(* CODESYS project TcDynCollections.library
   Company: FisoThemes
   DefaultNamespace: TcDynCollections
   Version: 1.0.5.27
   DocFormat: reStructuredText
   Placeholder: TwinCat Dynamic Collections
   Author: Goodwill Mzumala
   Description: A library for handling collections of data dynamically in TwinCAT.
   Title: TwinCat Dynamic Collections

Project tree, tasks and I/O mapping:
  libraries: Tc2_Standard, * (Beckhoff Automation GmbH); Tc2_System, * (Beckhoff Automation GmbH); Tc2_Utilities, 3.3.38.0 (Beckhoff Automation GmbH); Tc3_Module, * (Beckhoff Automation GmbH)
  DUTs/
    Aliases/
      data type T_AVL_Map_Node
      data type T_AVL_Node
      data type T_BST_Traversal
      data type T_Capacity
      data type T_Comparison
      data type T_Error
      data type T_Generic
      data type T_Hashmap_Bucket_Node
      data type T_Hashset_Bucket_Node
      data type T_List_Node
      data type T_Map_Entry
      data type T_Position
      data type T_Type
    Enums/
      data type E_BINARY_SEARCH_TREE_TRAVERSAL
      data type E_COMPARISON
      data type E_ERROR_CODE
    Structs/
      data type ST_AVL_MAP_NODE
      data type ST_AVL_NODE
      data type ST_ERROR
      data type ST_HASHMAP_BUCKET_NODE
      data type ST_HASHSET_BUCKET_NODE
      data type ST_LIST_NODE
      data type ST_MAP_ENTRY
      data type ST_ORDERED_HASHMAP_BUCKET_NODE
      data type ST_ORDERED_HASHSET_BUCKET_NODE
  GVLs/
    global variables GVL_Constants
    global variables GVL_Errors
  ITFs/
    Collections/
      Immutable/
        interface I_Immutable_Array: _Begin, _End, Contains, Get, Get_As_String, Get_Type_At, Search
        interface I_Immutable_Collection
        interface I_Immutable_List: _Begin, _End, Contains, Get, Get_As_String, Get_Type_At, Search
        interface I_Immutable_Map: Contains, Get, Get_As_String, Get_Keys, Get_Values
        interface I_Immutable_Set: Contains, Get_Values
      interface I_Array: _Begin, _End, Contains, Get, Get_As_String, Get_Generic, Get_Type_At, Reverse, Search, Set, Set_Generic, Swap
      interface I_Array_List: _Capacity
      interface I_Collection: _Count, _Empty, _Error_Status
      interface I_Deque: _Values, Back, Clear, Dequeue_At_Back, Dequeue_At_Front, Enqueue_At_Back, Enqueue_At_Front, Enqueue_Generic, Front, Reverse
      interface I_Hash_Map: _Bucket_Count, Resize
      interface I_Hash_Set: _Bucket_Count, Resize
      interface I_List: _Begin, _End, Append, Clear, Contains, Get, Get_As_String, Get_Generic, Get_Type_At, Insert, Insert_Generic, Prepend, Remove, Remove_At, Remove_Last, Resize, Reverse, Search, Set, Set_Generic, Swap
      interface I_Map: Clear, Contains, Get, Get_As_String, Get_Generic, Get_Keys, Get_Values, Insert, Insert_Generic, Remove, Remove_Generic, Update, Update_Generic, Upsert
      interface I_Queue: _Values, Clear, Dequeue, Enqueue, Enqueue_At_Front, Enqueue_Generic, Get, Get_Generic, Reverse
      interface I_Set: Clear, Contains, Get_Values, Insert, Insert_Generic, Remove, Remove_Generic
      interface I_Stack: _Values, Clear, Get, Get_Generic, Pop, Push, Push_Generic, Reverse
      interface I_Tree_Map: _Traversal
      interface I_Tree_Set: _Traversal
    Enumerators/
      interface I_Enumerable: Get_Enumerator
      interface I_Enumerator: Current, Current_As_String, Dispose, Next, Reset
    Iterable/
      interface I_Iterable: _Begin, _End
    Misc/
      interface I_Copyable: Copy_To
  POUs/
    Examples/
    Function Blocks/
      Collections/
        Immutable/
          function block FB_Immutable_Array [ST]: _Begin, _Count, _Empty, _End, _Error_Status, Contains, Get, Get_As_String, Get_Type_At, Search
          function block FB_Immutable_List [ST]: _Begin, _Count, _Empty, _End, _Error_Status, Contains, Get, Get_As_String, Get_Type_At, Search
          function block FB_Immutable_Map [ST]: _Count, _Empty, _Error_Status, Contains, Get, Get_As_String, Get_Keys, Get_Values
          function block FB_Immutable_Set [ST]: _Count, _Empty, _Error_Status, Contains, Get_Values
        function block FB_Array [ST]: _Begin, _End, Contains, FB_exit, FB_init, Get, Get_As_String, Get_Generic, Get_Type_At, Reverse, Search, Set, Set_Generic, Swap
        function block FB_Array_List [ST]: _Begin, _Capacity, _End, Append, Clear, Contains, FB_exit, FB_init, Get, Get_As_String, Get_Generic, Get_Type_At, Insert, Insert_Generic, Prepend, Remove, Remove_At, Remove_Last, Resize, Reverse, Search, Set, Set_Generic, Swap
        function block FB_Collection [ST]: Clear_Error, Decrement_Count, Increment_Count, _Count, _Empty, _Error_Status
        function block FB_Deque [ST]: _Count, _Empty, _Error_Status, _Values, Back, Clear, Dequeue_At_Back, Dequeue_At_Front, Enqueue_At_Back, Enqueue_At_Front, Enqueue_Generic, Front, Reverse
        function block FB_Hash_Map [ST]: Create_Buckets, Create_Node, Delete_Node, Hash, _Bucket_Count, Clear, Contains, FB_exit, FB_init, Get, Get_As_String, Get_Generic, Get_Keys, Get_Values, Insert, Insert_Generic, Remove, Remove_Generic, Resize, Update, Update_Generic, Upsert
        function block FB_Hash_Set [ST]: Create_Buckets, Create_Node, Delete_Node, Hash, _Bucket_Count, Clear, Contains, FB_exit, FB_init, Get_Values, Insert, Insert_Generic, Remove, Remove_Generic, Resize
        function block FB_List [ST]: Closest_Node_Iterator, Iterate, _Begin, _End, Append, Clear, Contains, FB_exit, Get, Get_As_String, Get_Generic, Get_Type_At, Insert, Insert_Generic, Prepend, Remove, Remove_At, Remove_Last, Resize, Reverse, Search, Set, Set_Generic, Swap
        function block FB_Queue [ST]: _Count, _Empty, _Error_Status, _Values, Clear, Dequeue, Enqueue, Enqueue_At_Front, Enqueue_Generic, Get, Get_Generic, Reverse
        function block FB_Stack [ST]: _Count, _Empty, _Error_Status, _Values, Clear, Get, Get_Generic, Pop, Push, Push_Generic, Reverse
        function block FB_Tree_Map [ST]: Balance, Clear_Node, Create_Node, Delete_Node, Find_Minimum_Node, Get_Balance, Get_Height, Move_Node, Remove_Node, Rotate_Left, Rotate_Right, Search_Node, Update_Height, _Traversal, Clear, Contains, FB_exit, Get, Get_As_String, Get_Generic, Get_Keys, Get_Values, Insert, Insert_Generic, Remove, Remove_Generic, Update, Update_Generic, Upsert
        function block FB_Tree_Multiset [ST]: Insert_Generic
        function block FB_Tree_Set [ST]: Balance, Clear_Node, Create_Node, Delete_Node, Find_Minimum_Node, Get_Balance, Get_Height, Move_Node, Remove_Node, Rotate_Left, Rotate_Right, Search_Node, Update_Height, _Traversal, Clear, Contains, FB_exit, Get_Values, Insert, Insert_Generic, Remove, Remove_Generic
      Enumerators/
        function block FB_Enumerator [ST]: Current, Current_As_String, Dispose, FB_exit, FB_init, Next, Reset
      Misc/
        function block FB_Free [ST]: FB_exit, FB_init
      Specialised/
      Wrappers/
    Functions/
      function F_Any_To_Generic [ST]
      function F_Clone_Generic [ST]
      function F_Compare_Any [ST]
      function F_Compare_Generics [ST]
      function F_Copy_Generic_Value [ST]
      function F_Delete_Generic [ST]
      function F_Error [ST]
      function F_Generic_To_DT [ST]
      function F_Generic_To_LREAL [ST]
      function F_Generic_To_LTIME [ST]
      function F_Generic_To_String [ST]
      function F_Is_Date_Generic [ST]
      function F_Is_Numeric_Generic [ST]
      function F_Is_Time_Generic [ST]
      function F_Malloc_Generic [ST]
      function F_Matching_Generics [ST]
      function F_Murmur_Scramble [ST]
      function F_Murmur3_Hash [ST]
      function F_String_Convertable_Generic [ST]
      function F_String_To_Any [ST]
      function F_Swap_Generics [ST]
    program MAIN [ST]
  Project Information/
    function F_GetCompany [ST]
    function F_GetTitle [ST]
    function F_GetVersion [ST]
  UML/
    Collections Interfaces
  Version/
    global variables Global_Version
  VISUs/
*)

// DUTs/Aliases/T_AVL_Map_Node
TYPE T_AVL_Map_Node : ST_AVL_MAP_NODE; END_TYPE

// DUTs/Aliases/T_AVL_Node
TYPE T_AVL_Node : ST_AVL_NODE; END_TYPE

// DUTs/Aliases/T_BST_Traversal
TYPE T_BST_Traversal : E_BINARY_SEARCH_TREE_TRAVERSAL; END_TYPE

// DUTs/Aliases/T_Capacity
TYPE T_Capacity : DINT(GVL_Constants.MIN_CAPACITY..GVL_Constants.MAX_CAPACITY); END_TYPE

// DUTs/Aliases/T_Comparison
TYPE T_Comparison : E_COMPARISON; END_TYPE

// DUTs/Aliases/T_Error
TYPE T_Error : ST_ERROR; END_TYPE

// DUTs/Aliases/T_Generic
TYPE T_Generic : __SYSTEM.AnyType; END_TYPE

// DUTs/Aliases/T_Hashmap_Bucket_Node
TYPE T_Hashmap_Bucket_Node : ST_HASHMAP_BUCKET_NODE; END_TYPE

// DUTs/Aliases/T_Hashset_Bucket_Node
TYPE T_Hashset_Bucket_Node : ST_HASHSET_BUCKET_NODE; END_TYPE

// DUTs/Aliases/T_List_Node
TYPE T_List_Node : ST_LIST_NODE; END_TYPE

// DUTs/Aliases/T_Map_Entry
TYPE T_Map_Entry : ST_MAP_ENTRY; END_TYPE

// DUTs/Aliases/T_Position
TYPE T_Position : DINT; END_TYPE

// DUTs/Aliases/T_Type
TYPE T_Type : __SYSTEM.TYPE_CLASS; END_TYPE

// DUTs/Enums/E_BINARY_SEARCH_TREE_TRAVERSAL
// Methods for traversing a binary search tree.
{attribute 'qualified_only'}
{attribute 'to_string'}
TYPE E_BINARY_SEARCH_TREE_TRAVERSAL :
(
	In_Order := 0,
	Pre_Order,
	Post_Order, 
	Level_Order
)BYTE;
END_TYPE

// DUTs/Enums/E_COMPARISON
// Comparison enum.
{attribute 'qualified_only'}
{attribute 'strict'}
{attribute 'to_string'}
TYPE E_COMPARISON :
(
	Invalid := 0,
	Less,
	Equal,
	Greater
)BYTE;
END_TYPE

// DUTs/Enums/E_ERROR_CODE
 // Error code are @ CmpErrors.Errors.<variable> from the CmpErrors2 Interfaces library.
 // https://help.codesys.com/webapp/Errors;product=CmpErrors2_Itfs;version=3.5.15.0
{attribute 'qualified_only'}
{attribute 'to_string'}
TYPE E_ERROR_CODE :
(
	ERR_OK 						 := 16#0,	//	Ok
	ERR_FAILED 					 := 16#1, 	//	General error - To be used only for internal errors
	ERR_PARAMETER 				 := 16#2, 	//	Invalid parameter for this operation
	ERR_NOT_INITIALIZED 		 := 16#3, 	//	Function cannot be executed, since component has not been initialized yet. It may work later, though
	ERR_VERSION 				 := 16#4, 	//	Version conflict
	ERR_TIMEOUT 				 := 16#5, 	//	Operation timed out
	ERR_NO_BUFFER 				 := 16#6, 	//	Insufficient memory to carry out the request
	ERR_PENDING 				 := 16#A, 	//	For async-calls: call not complete, yet
	ERR_NUM_PENDING 			 := 16#B, 	//  Too many pending calls. Try later
	ERR_NOT_IMPLEMENTED 		 := 16#C, 	//  The function is not implemented
	ERR_INVALID_ID 				 := 16#D, 	//  No object with the provided id found
	ERR_OVERFLOW 				 := 16#E, 	//	Integer overflow
	ERR_BUFFER_SIZE 			 := 16#F, 	//	The size of a buffer is too small OR invalid
	ERR_NO_OBJECT 				 := 16#10,	//	No object with this specified name available
	ERR_NO_MEMORY 				 := 16#11,	//  No heap memory available
	ERR_DUPLICATE 				 := 16#12A, //  An object with the same name is still available
	ERR_MEMORY_OVERWRITE 		 := 16#13,  //  Heap memory was written out of bounds! Memory overwrite error
	ERR_INVALID_HANDLE 			 := 16#14,  //  Invalid handle to an object
	ERR_END_OF_0BJECT 			 := 16#15,  //  End OF object reached
	ERR_NO_CHANGE 				 := 16#16,  //  No changes done
	ERR_INVALID_INTERFACE 		 := 16#17,  //  Invalid or unknown interface
	ERR_NOT_SUPPORTED 			 := 16#18,  //  Functionality not supported
	ERR_NO_ACCESS_RIGHTS 		 := 16#19,  //  No access rights for this operation
	ERR_OUT_OF_LIMITS 			 := 16#1A,  //  Specified limits of a resource exceeded
	ERR_ENTRIES_REMAINING 		 := 16#1B,  //  Remaining entries that could not be transmitted because of buffer limitation
	ERR_INVALID_SESSION_ID 		 := 16#1C,  //  Invalid online sessionid
	ERR_EXCEPTION 				 := 16#1D,  //  Exception occurred
	ERR_SIGNATURE_MISMATCH 		 := 16#1E,	//	Signature mismatch of an api function
	ERR_VERSION_MISMATCH 		 := 16#1F,	//	Version mismatch
	ERR_TYPE_MISMATCH 			 := 16#20,	//	Type mismatch
	ERR_ID_MISMATCH 			 := 16#21,	//	ID mismatch
	ERR_NO_CONSISTENCY 			 := 16#22,	//	Consistency error
	ERR_NO_COMM_CYCLE 			 := 16#23,	//	No COMM_CYCLE needed
	ERR_DONT_SUSPEND_TASK 		 := 16#24,	//	Do not suspend task after an exception
	ERR_MEMORY_LOCK_FAILED 		 := 16#25,	//	Memory cannot be locked in this operation
	ERR_LICENSE_MISSING 		 := 16#26,	//	License missing for the runtime
	ERR_OPERATION_DENIED 		 := 16#27,	//	Operation denied 
	ERR_DEVICE 					 := 16#28,	//	Device error
	ERR_DISK_FULL 				 := 16#29,	//	Disk full
	ERR_CRC_FAILED 				 := 16#30,	//	Internal use in runtime
	ERR_MEDIA_ERASE 			 := 16#31,	//	Internal use in runtime
	ERR_FILE_ERROR 				 := 16#32,	//	File error. e.g. cannot open a file for writing because it could be write protected
	ERR_NO_RETAIN_MEMORY 		 := 16#33,	//	No retain memory available
	ERR_OUT_OF_LIMITS_MIN 		 := 16#34,	//	Specified minimum-limit of a resource exceeded
	ERR_OUT_OF_LIMITS_MAX 		 := 16#35,	//	Specified maximum-limit of a resource exceeded
	ERR_SIZE_MISMATCH 			 := 16#36,	//	Size mismatch
	ERR_CALL_AGAIN 				 := 16#37,	//	Operation is not yet finished, call function again to proceed
	ERR_NOTHING_TO_DO 			 := 16#38,	//	Operation has nothing to do. No execution.
	ERR_SECURITY_CHECKS_FAILED 	 := 16#39,	//	Some security checks have failed. /* This is a generic error code to report this error over public channels. In this case the error code doesn’t provide a detailed cause for the error. */
	ERR_INVALID_SEQUENCE 		 := 16#3A,	//	 
	ERR_INVALID_REFERENCE 		 := 16#3B,	//	Dereferencing an IEC reference in IecVarAccess failed due to invalid destination address, e. G. NULL.
	ERR_CONVERSION_INCOMPLETE 	 := 16#3C,	//	Conversion of string encodings was not lossless.
	ERR_SOCK_NOT_INITIALIZED 	 := 16#201, //  Socket errors (range: 0x0200 - 0X02FF)
	ERR_SOCK_NOT_SOCKET 		 := 16#202, //  The provided socket handle is invalid
	ERR_SOCK_AF_UNSUPPORTED 	 := 16#203, //  The address family is not supported
	ERR_SOCK_PROTO_UNSUPPORTED   := 16#204, //  Protocol is not supported */
	ERR_SOCK_NO_BUFFER 			 := 16#205, //  Not enough buffer to handle the request */
	ERR_SOCK_WOULD_BLOCK 		 := 167206, //  Socket is in nonblocking mode but this call would block =/
	ERR_SOCK_ADDR_INUSE 		 := 16#207, //  The provided address is already in use */
	ERR_SOCK_ADDR_NOT_AVAILABLE  := 16#208, //  The provided address is not available on THIS computer */
	ERR_SOCK_CONN_REFUSED 		 := 16#209, //  Connection has been refused by the remote host */
	ERR_SOCK_TIMEDOUT 			 := 16#20A, //  Operation timed out */
	ERR_SOCK_HOST_NOT_FOUND 	 := 16#20B, //  The host has NOT been found */
	ERR_SOCK_HOST_UNREACHABLE  	 := 16#20C, //  Host is unreachable */
	ERR_SOCK_1S_CONNECTED 		 := 16#20D, //  Socket is already connected =/
	ERR_SOCK_NOT_CONNECTED 		 := 16#20E, //  The socket is not connected */
	ERR_SOCK_SHUTDOWN 			 := 16#20F, //  Shutdown has been called on the socket =/
	ERR_SOCK_MSGSIZE 			 := 16#210, //  For sockets of type DGRAM. The package to send exceeds the maximum package size =/
	ERR_SOCK_CLOSED 			 := 16#211, //  Socket has been gracefully closed. No more send/receives allowed =/
	ERR_L7_TAG_MISSING 			 := 16#300,	//  Tag missing in online communication buffer
	ERR_L7_UNKNOWN_CMD_GROUP 	 := 16#301,	//  Unknown command group
	ERR_L7_UNKNOWN_CMD 			 := 16#302,	//  Unknown command (within a valid command group)
	ERR_L7_INCOMPLETE 			 := 16#303	//  Level 7 service incomplete
)DINT;
END_TYPE

// DUTs/Structs/ST_AVL_MAP_NODE
// Node for an AVL Tree Map.
{attribute 'enable_dynamic_creation'}
TYPE ST_AVL_MAP_NODE EXTENDS ST_MAP_ENTRY :
STRUCT
	Height 		: T_Position; // Height of the node.
	pParent 	: POINTER TO ST_AVL_MAP_NODE; 	// Pointer to parent node.
	pLeft 		: POINTER TO ST_AVL_MAP_NODE; 	// Pointer to left node.
	pRight 		: POINTER TO ST_AVL_MAP_NODE; 	// Pointer to right node.
END_STRUCT
END_TYPE

// DUTs/Structs/ST_AVL_NODE
// Node for AVL Tree.
{attribute 'enable_dynamic_creation'}
TYPE ST_AVL_NODE:
STRUCT
	Data 		: T_Generic; // Stored data.
	Height 		: T_Position; // Height of the node.
	pParent 	: POINTER TO ST_AVL_NODE; 	// Pointer to parent node.
	pLeft 		: POINTER TO ST_AVL_NODE; 	// Pointer to left node.
	pRight 		: POINTER TO ST_AVL_NODE; 	// Pointer to right node.
END_STRUCT
END_TYPE

// DUTs/Structs/ST_ERROR
// STRUCT used to contain error status information.
{attribute 'enable_dynamic_creation'}
TYPE ST_ERROR :
STRUCT
	nCODE 	: DINT; // Error code specific to the particular error.
	bSTATUS : BOOL; // Indicates if an error has occurred | TRUE = error, FALSE = no error
	sSOURCE : STRING; // Textual information describing the error.
END_STRUCT
END_TYPE

// DUTs/Structs/ST_HASHMAP_BUCKET_NODE
{attribute 'enable_dynamic_creation'}
TYPE ST_HASHMAP_BUCKET_NODE EXTENDS ST_MAP_ENTRY :
STRUCT
	pNext : POINTER TO ST_HASHMAP_BUCKET_NODE;
END_STRUCT
END_TYPE

// DUTs/Structs/ST_HASHSET_BUCKET_NODE
{attribute 'enable_dynamic_creation'}
TYPE ST_HASHSET_BUCKET_NODE :
STRUCT
	Data : T_Generic;
	pNext : POINTER TO ST_HASHSET_BUCKET_NODE;
END_STRUCT
END_TYPE

// DUTs/Structs/ST_LIST_NODE
// Node for linked list.
{attribute 'enable_dynamic_creation'}
TYPE ST_LIST_NODE:
STRUCT
	Data 		: T_Generic; // Stored data.
	pPrevious 	: POINTER TO ST_LIST_NODE; 	// Pointer to previous node.
	pNext 		: POINTER TO ST_LIST_NODE; 	// Pointer to next node.
END_STRUCT
END_TYPE

// DUTs/Structs/ST_MAP_ENTRY
// Entry for a key value pair.
{attribute 'enable_dynamic_creation'}
TYPE ST_MAP_ENTRY :
STRUCT
	Key : T_Generic; // Key used to identify stored value    
	Value : T_Generic; // Value to store in dictionary with key
END_STRUCT
END_TYPE

// DUTs/Structs/ST_ORDERED_HASHMAP_BUCKET_NODE
{attribute 'enable_dynamic_creation'}
TYPE ST_ORDERED_HASHMAP_BUCKET_NODE EXTENDS ST_MAP_ENTRY:
STRUCT
	pNext,
	pBefore,
	pAfter 	: POINTER TO ST_ORDERED_HASHSET_BUCKET_NODE;
END_STRUCT
END_TYPE

// DUTs/Structs/ST_ORDERED_HASHSET_BUCKET_NODE
{attribute 'enable_dynamic_creation'}
TYPE ST_ORDERED_HASHSET_BUCKET_NODE :
STRUCT
	Data 	: T_Generic;
	pNext,
	pBefore,
	pAfter 	: POINTER TO ST_ORDERED_HASHSET_BUCKET_NODE;
END_STRUCT
END_TYPE

// GVLs/GVL_Constants
{attribute 'qualified_only'}
VAR_GLOBAL CONSTANT
	MIN_CAPACITY : DINT := 0;
	MAX_CAPACITY : DINT := 2147483647;
END_VAR

// GVLs/GVL_Errors
// Library errors
{attribute 'qualified_only'}
VAR_GLOBAL CONSTANT
	ERR_NO_ERROR 			: T_Error := (bStatus := FALSE,	nCode := E_ERROR_CODE.ERR_OK, 				sSource := 'No Error.'); // No Error.
	ERR_TYPE_MISMATCH 		: T_Error := (bStatus := TRUE,	nCode := E_ERROR_CODE.ERR_TYPE_MISMATCH, 	sSource := 'Type mismatch.'); // Type mismatch.
	ERR_SIZE_MISMATCH 		: T_Error := (bStatus := TRUE,	nCode := E_ERROR_CODE.ERR_SIZE_MISMATCH, 	sSource := 'Size mismatch.'); // Size mismatch.
	ERR_INVALID_REFERENCE 	: T_Error := (bStatus := TRUE,	nCode := E_ERROR_CODE.ERR_INVALID_REFERENCE,sSource := 'Invalid reference.'); // Invalid reference.
	ERR_INVALID_INTERFACE 	: T_Error := (bStatus := TRUE,	nCode := E_ERROR_CODE.ERR_INVALID_INTERFACE,sSource := 'Invalid interface.'); // Invalid interface.
	ERR_INVALID_CONVERSION	: T_Error := (bStatus := TRUE,	nCode := E_ERROR_CODE.ERR_NOT_SUPPORTED, 	sSource := 'Conversion not supported.'); // Conversion not supported.
	ERR_INVALID_COMPARISON	: T_Error := (bStatus := TRUE,	nCode := E_ERROR_CODE.ERR_NOT_SUPPORTED, 	sSource := 'Invalid comparison.'); // Invalid comparison.
	ERR_NO_KEY 				: T_Error := (bStatus := TRUE,	nCode := E_ERROR_CODE.ERR_NO_OBJECT,		sSource := 'Key not found.'); // Key not found.'
	ERR_NO_ITEM 			: T_Error := (bStatus := TRUE,	nCode := E_ERROR_CODE.ERR_NO_OBJECT, 		sSource := 'Item not found.'); // Item not found.
	ERR_INDEX_OUT_OF_BOUNDS : T_Error := (bStatus := TRUE,	nCode := E_ERROR_CODE.ERR_OUT_OF_LIMITS, 	sSource := 'Index out of bounds.'); // Index out of bounds.
	ERR_DUPLICATE_KEY 		: T_Error := (bStatus := TRUE,	nCode := E_ERROR_CODE.ERR_DUPLICATE, 		sSource := 'Duplicate key.'); // Duplicate key.
	ERR_DUPLICATE_ITEM 		: T_Error := (bStatus := TRUE,	nCode := E_ERROR_CODE.ERR_DUPLICATE, 		sSource := 'Duplicate item.'); // Duplicate item.
	ERR_MALLOC_FAILED 		: T_Error := (bStatus := TRUE,	nCode := E_ERROR_CODE.ERR_NO_MEMORY, 		sSource := 'Memory allocation failed.'); // Memory allocation failed.
END_VAR

// Version/Global_Version
{attribute 'TcGenerated'}
{attribute 'no-analysis'}
{attribute 'linkalways'}
// This function has been automatically generated from the project information.
VAR_GLOBAL CONSTANT
	{attribute 'const_non_replaced'}
	stLibVersion_TwinCat_Dynamic_Collections : ST_LibVersion := (iMajor := 1, iMinor := 0, iBuild := 5, iRevision := 27, nFlags := 0, sVersion := '1.0.5.27');
END_VAR

// ITFs/Collections/Immutable/I_Immutable_Array
// Interface for an immutable array.
INTERFACE I_Immutable_Array EXTENDS I_Immutable_Collection

// Index of the first element.
PROPERTY _Begin : T_Position
GET
END_GET
END_PROPERTY

// Index of the last element.
PROPERTY _End : T_Position
GET
END_GET
END_PROPERTY

// Checks if item is contained in array.
METHOD Contains : BOOL
VAR_INPUT
	Item : ANY; // Item to find.
END_VAR
END_METHOD

// Gets item from array at specified location.
METHOD Get : I_Immutable_Array
VAR_INPUT
	Index : T_Position; // Location of item.
	Item : ANY;  // Variable to store returned item.
END_VAR
VAR_OUTPUT
	bSuccess : BOOL;
END_VAR
END_METHOD

// Returns item as a string, if type to string conversion is supported.
METHOD Get_As_String : I_Immutable_Array
VAR_INPUT
	Index : T_Position; // Location of item.
	sItem : REFERENCE TO STRING; // Variable to store returned item.
END_VAR
VAR_OUTPUT
	bSuccess : BOOL;
END_VAR
END_METHOD

// Gets the type of the item at specified location.
METHOD Get_Type_At : I_Immutable_Array
VAR_INPUT
	Index : T_Position;
END_VAR
VAR_OUTPUT
	Item_Type : T_Type;
	bSuccess : BOOL;
END_VAR
END_METHOD

// Find the location of an item in the array.
METHOD Search : I_Immutable_Array
VAR_INPUT
	Item : ANY; // Item to find.
END_VAR
VAR_OUTPUT
	Index : T_Position; //Location of item.
	bSuccess : BOOL;
END_VAR
END_METHOD

END_INTERFACE

// ITFs/Collections/Immutable/I_Immutable_Collection
// Base interface for immutable collections
INTERFACE I_Immutable_Collection EXTENDS I_Collection

END_INTERFACE

// ITFs/Collections/I_Collection
// Base interface for collections.
INTERFACE I_Collection EXTENDS __SYSTEM.IQueryInterface

// Number of items in the collection.
PROPERTY _Count : T_Capacity
GET
END_GET
END_PROPERTY

// Checks if collection is empty.
PROPERTY _Empty : BOOL
GET
END_GET
END_PROPERTY

// Error status of the collection.
PROPERTY _Error_Status : T_Error
GET
END_GET
END_PROPERTY

END_INTERFACE

// ITFs/Collections/Immutable/I_Immutable_List
// Interface for an immutable list.
INTERFACE I_Immutable_List EXTENDS I_Immutable_Collection

// Index of the first element.
PROPERTY _Begin : T_Position
GET
END_GET
END_PROPERTY

// Index of the last element.
PROPERTY _End : T_Position
GET
END_GET
END_PROPERTY

(* Checks if item is contained in list *)
METHOD Contains : BOOL
VAR_INPUT
	Item : ANY; // Item to find in list
END_VAR
END_METHOD

// Gets item from list at specified location without removing it.
METHOD Get : I_Immutable_List
VAR_INPUT
	Index : T_Position; // Location of item
	Item : ANY;  // Variable to store returned item
END_VAR
VAR_OUTPUT
	bSuccess : BOOL;
END_VAR
END_METHOD

// Returns item as a string, if type to string conversion is supported.
METHOD Get_As_String : I_Immutable_List
VAR_INPUT
	Index : T_Position; // Location of item
	sItem : REFERENCE TO STRING; // Variable to store returned item.
END_VAR
VAR_OUTPUT
	bSuccess : BOOL;
END_VAR
END_METHOD

// Gets the type of the item at specified location.
METHOD Get_Type_At : I_Immutable_List
VAR_INPUT
	Index : T_Position;
END_VAR
VAR_OUTPUT
	Item_Type : T_Type;
	bSuccess : BOOL;
END_VAR
END_METHOD

// Find the location of an item in list.
METHOD Search : I_Immutable_List
VAR_INPUT
	Item : ANY; // Item to find in list
END_VAR
VAR_OUTPUT
	Index : T_Position; //Location of item in list 
	bSuccess : BOOL;
END_VAR
END_METHOD

END_INTERFACE

// ITFs/Collections/Immutable/I_Immutable_Map
INTERFACE I_Immutable_Map EXTENDS I_Immutable_Collection

// Checks if key is contained in the map.
METHOD Contains : BOOL
VAR_INPUT
	Key : ANY; // Key to find.
END_VAR
END_METHOD

// Gets the value associated with the specified key without removing it from the map.
METHOD Get : I_Immutable_Map
VAR_INPUT
	Key : ANY; // Key used to identify stored value
	Value : ANY; // Variable to store requested data 
END_VAR
VAR_OUTPUT
	bSuccess : BOOL;
END_VAR
END_METHOD

// Returns value as a string, if type to string conversion is supported.
METHOD Get_As_String : I_Immutable_Map
VAR_INPUT
	Key : ANY; // Key used to identify stored value
	sValue : REFERENCE TO STRING; // Variable to store returned item.
END_VAR
VAR_OUTPUT
	bSuccess : BOOL;
END_VAR
END_METHOD

// Gets an immutable list of the keys.
METHOD Get_Keys : I_Immutable_List
VAR_INPUT
END_VAR
END_METHOD

// Gets an immutable list of the values.
METHOD Get_Values : I_Immutable_List
VAR_INPUT
END_VAR
END_METHOD

END_INTERFACE

// ITFs/Collections/Immutable/I_Immutable_Set
// Interface for immutable set.
INTERFACE I_Immutable_Set EXTENDS I_Immutable_Collection

// Checks if item is contained in set.
METHOD Contains : BOOL
VAR_INPUT
	Item : ANY; // Item to find.
END_VAR
END_METHOD

// Gets an immutable list of the values in the set.
METHOD Get_Values : I_Immutable_List
END_METHOD

END_INTERFACE

// ITFs/Collections/I_Array
// Interface for a static array.
INTERFACE I_Array EXTENDS I_Collection

// Index of the first element.
PROPERTY _Begin : T_Position
GET
END_GET
END_PROPERTY

// Index of the last element.
PROPERTY _End : T_Position
GET
END_GET
END_PROPERTY

// Checks if item is contained in array.
METHOD Contains : BOOL
VAR_INPUT
	Item : ANY; // Item to find.
END_VAR
END_METHOD

// Gets item from array at specified location.
METHOD Get : I_Array
VAR_INPUT
	Index : T_Position; // Location of item.
	Item : ANY;  // Variable to store returned item.
END_VAR
VAR_OUTPUT
	bSuccess : BOOL;
END_VAR
END_METHOD

// Returns item as a string, if type to string conversion is supported.
METHOD Get_As_String : I_Array
VAR_INPUT
	Index : T_Position; // Location of item.
	sItem : REFERENCE TO STRING; // Variable to store returned item.
END_VAR
VAR_OUTPUT
	bSuccess : BOOL;
END_VAR
END_METHOD

// Gets an item from the array in it's generic form.
// (** Use carefully as this contains the pointer of the actual value in the collection. **)
// If you wish to use this it is recommeded you create a copy of the returned value using MEMMOVE or MEMCPY
METHOD Get_Generic : I_Array
VAR_INPUT
	Index : T_Position; // Location of item.
END_VAR
VAR_OUTPUT
	Item : T_Generic;
	bSuccess : BOOL;
END_VAR
END_METHOD

// Gets the type of the item at specified location.
METHOD Get_Type_At : I_Array
VAR_INPUT
	Index : T_Position;
END_VAR
VAR_OUTPUT
	Item_Type : T_Type;
	bSuccess : BOOL;
END_VAR
END_METHOD

// Reverses the order of items in the array.
METHOD Reverse : I_Array
VAR_OUTPUT
	bSuccess : BOOL;
END_VAR
END_METHOD

// Find the location of an item in the array.
METHOD Search : I_Array
VAR_INPUT
	Item : ANY; // Item to find.
END_VAR
VAR_OUTPUT
	Index : T_Position; //Location of item.
	bSuccess : BOOL;
END_VAR
END_METHOD

// Changes the item at the specified location in the array.
METHOD Set : I_Array
VAR_INPUT
	Index 	: T_Position; // Location of item.
	Item 	: ANY; 	// Item to store.
END_VAR
VAR_OUTPUT
	bSuccess : BOOL;
END_VAR
END_METHOD

// Changes the item at the specified location in the array in it's generic form.
METHOD Set_Generic : I_Array
VAR_INPUT
	Index : T_Position; // Location of item.
	Item : T_Generic; // Item to store.
END_VAR
VAR_OUTPUT
	bSuccess : BOOL;
END_VAR
END_METHOD

// Swaps item at index with item at index B.
METHOD Swap : I_Array
VAR_INPUT
	Index_A, Index_B : T_Position;
END_VAR
VAR_OUTPUT
	bSuccess : BOOL;
END_VAR
END_METHOD

END_INTERFACE

// ITFs/Collections/I_Array_List
// Interface for the array list.
INTERFACE I_Array_List EXTENDS I_List

// Size of the storage space currently allocated for the array list.
PROPERTY _Capacity : T_Capacity
GET
END_GET
END_PROPERTY

END_INTERFACE

// ITFs/Collections/I_List
// Interface for a list.
INTERFACE I_List EXTENDS I_Collection

// Index of the first element.
PROPERTY _Begin : T_Position
GET
END_GET
END_PROPERTY

// Index of the last element.
PROPERTY _End : T_Position
GET
END_GET
END_PROPERTY

// Adds an item to the end of the list.
METHOD Append : I_List
VAR_INPUT
	Item : ANY; // Value to store in list
END_VAR
VAR_OUTPUT
	bSuccess : BOOL;
END_VAR
END_METHOD

// Empties/Clears/Deletes every item in the list.
METHOD Clear : I_List
END_METHOD

// Checks if item is contained in list.
METHOD Contains : BOOL
VAR_INPUT
	Item : ANY; // Item to find in list
END_VAR
END_METHOD

// Gets item from list at specified location without removing it
METHOD Get : I_List
VAR_INPUT
	Index : T_Position; // Location of item
	Item : ANY;  // Variable to store returned item
END_VAR
VAR_OUTPUT
	bSuccess : BOOL;
END_VAR
END_METHOD

// Returns item as a string, if type to string conversion is supported
METHOD Get_As_String : I_List
VAR_INPUT
	Index : T_Position; // Location of item
	sItem : REFERENCE TO STRING; // Variable to store returned item.
END_VAR
VAR_OUTPUT
	bSuccess : BOOL;
END_VAR
END_METHOD

// Gets a value from a list in it's generic form.
// (** Use carefully as this contains the pointer of the actual value in the collection. **)
// If you wish to use this it is recommeded you create a copy of the returned value using MEMMOVE or MEMCPY
METHOD Get_Generic : I_List
VAR_INPUT
	Index : T_Position; // Location of item
END_VAR
VAR_OUTPUT
	Item : T_Generic;
	bSuccess : BOOL;
END_VAR
END_METHOD

// Gets the type of the item at specified location.
METHOD Get_Type_At : I_List
VAR_INPUT
	Index : T_Position;
END_VAR
VAR_OUTPUT
	Item_Type : T_Type;
	bSuccess : BOOL;
END_VAR
END_METHOD

// Adds new item to list at specified location, if index = 0, item will be added at the front, if index = count, item will be added at the back
METHOD Insert : I_List
VAR_INPUT
	Index : T_Position; // Location of item
	Item : ANY; // Item to store in list
END_VAR
VAR_OUTPUT
	bSuccess : BOOL;
END_VAR
END_METHOD

// Adds new item to list at specified location using the generic form. 
// If index = 0, item will be added at the front, if index = count, item will be added at the back
METHOD Insert_Generic : I_List
VAR_INPUT
	Index 	 : T_Position; 	// Location of item
	Item 	 : T_Generic;  	// Item to store in list
END_VAR
VAR_OUTPUT
	bSuccess : BOOL;
END_VAR
END_METHOD

// Adds an item at the front of the list.
METHOD Prepend : I_List
VAR_INPUT
	Item : ANY; // Value to store in list
END_VAR
VAR_OUTPUT
	bSuccess : BOOL;
END_VAR
END_METHOD

// Removes item from the list.
METHOD Remove : I_List
VAR_INPUT
	Item : ANY; // Item to remove from in list
END_VAR
VAR_OUTPUT
	bSuccess : BOOL;
END_VAR
END_METHOD

// Remove item at specified location 
METHOD Remove_At : I_List
VAR_INPUT
	Index : T_Position; // Location of item
END_VAR
VAR_OUTPUT
	bSuccess : BOOL;
END_VAR
END_METHOD

// Removes item at the back of the list.
METHOD Remove_Last : I_List
VAR_OUTPUT
	bSuccess : BOOL;
END_VAR
END_METHOD

// Manually resize list. If list becomes smaller, item on higher locations will be deleted.
METHOD Resize : I_List
VAR_INPUT
	Size : T_Capacity; // New size of list.
END_VAR
VAR_OUTPUT
	bSuccess : BOOL;
END_VAR
END_METHOD

// Reverses the order of items in the list
METHOD Reverse : I_List
VAR_OUTPUT
	bSuccess : BOOL;
END_VAR
END_METHOD

// Find the location of an item in list.
METHOD Search : I_List
VAR_INPUT
	Item : ANY; // Item to find in list
END_VAR
VAR_OUTPUT
	Index : T_Position; //Location of item in list 
	bSuccess : BOOL;
END_VAR
END_METHOD

// Changes the item at the specified location in the list.
METHOD Set : I_List
VAR_INPUT
	Index 	: T_Position; // Location of item
	Item 	: ANY; 	// Item to store in list
END_VAR
VAR_OUTPUT
	bSuccess : BOOL;
END_VAR
END_METHOD

// Changes the item at the specified location in the list in it's generic form.
METHOD Set_Generic : I_List
VAR_INPUT
	Index : T_Position; // Location of item
	Item : T_Generic; // Item to store in list
END_VAR
VAR_OUTPUT
	bSuccess : BOOL;
END_VAR
END_METHOD

// Swaps item at index A with item at index B.
METHOD Swap : I_List
VAR_INPUT
	Index_A, Index_B : T_Position;
END_VAR
VAR_OUTPUT
	bSuccess : BOOL;
END_VAR
END_METHOD

END_INTERFACE

// ITFs/Collections/I_Deque
// Interface for a double ended queue - Deque
INTERFACE I_Deque EXTENDS I_Collection

// Gets an immutable list of the items in Deque.
PROPERTY _Values : I_Immutable_List
GET
END_GET
END_PROPERTY

// Get item at the back of the deque without removing it.
METHOD Back : I_Deque
VAR_INPUT
	Item : ANY; // Variable to store returned item value
END_VAR
VAR_OUTPUT
	bSuccess : BOOL;
END_VAR
END_METHOD

// Empties/Clears/Deletes every item in the deque.
METHOD Clear : I_Deque
END_METHOD

// Removes item at the front of the deque.
METHOD Dequeue_At_Back : I_Deque
VAR_OUTPUT
	bSuccess : BOOL;
END_VAR
END_METHOD

// Removes item at the front of the deque.
METHOD Dequeue_At_Front : I_Deque
VAR_OUTPUT
	bSuccess : BOOL;
END_VAR
END_METHOD

// Adds item at the back of the deque.
METHOD Enqueue_At_Back : I_Deque
VAR_INPUT
	Item : ANY; // Item to store.
END_VAR
VAR_OUTPUT
	bSuccess : BOOL;
END_VAR
END_METHOD

// Add item to the front of the deque.
METHOD Enqueue_At_Front : I_Deque
VAR_INPUT
	Item : ANY; // Item to store.
END_VAR
VAR_OUTPUT
	bSuccess : BOOL;
END_VAR
END_METHOD

// Adds a generic item at the back of the deque.
METHOD Enqueue_Generic : I_Deque
VAR_INPUT
	Item : T_Generic; // Item to store.
	bAt_Front : BOOL; // Enqueues at front if set to TRUE.
END_VAR
VAR_OUTPUT
	bSuccess : BOOL;
END_VAR
END_METHOD

// Get item at the front of the deque without removing it.
METHOD Front : I_Deque
VAR_INPUT
	Item : ANY; // Variable to store returned item value
END_VAR
VAR_OUTPUT
	bSuccess : BOOL;
END_VAR
END_METHOD

// Reverses the order of items in the deque.
METHOD Reverse : I_Deque
VAR_OUTPUT
	bSuccess : BOOL;
END_VAR
END_METHOD

END_INTERFACE

// ITFs/Collections/I_Hash_Map
// Interface for a set implemented using a hash table.
INTERFACE I_Hash_Map EXTENDS I_Map

// Number of buckets in the hash map.
PROPERTY _Bucket_Count : T_Capacity;
GET
END_GET
END_PROPERTY

// Sets the number of buckets in the hash map.
// Existing items are rehashed and redistributed into the new buckets.
METHOD Resize : I_Hash_Map
VAR_INPUT
	Count : T_Capacity;
END_VAR
VAR_OUTPUT
	bSuccess : BOOL;
END_VAR
END_METHOD

END_INTERFACE

// ITFs/Collections/I_Map
// An interface for a collection that holds key/value pairs  
INTERFACE I_Map EXTENDS I_Collection

// Empties/Clears/Deletes every item in the map.
METHOD Clear : I_Map
END_METHOD

// Checks if key is contained in the map.
METHOD Contains : BOOL
VAR_INPUT
	Key : ANY; // Key to find.
END_VAR
END_METHOD

// Gets the value associated with the specified key without removing it from the map.
METHOD Get : I_Map
VAR_INPUT
	Key : ANY; // Key used to identify stored value
	Value : ANY; // Variable to store requested data 
END_VAR
VAR_OUTPUT
	bSuccess : BOOL;
END_VAR
END_METHOD

// Returns value as a string, if type to string conversion is supported.
METHOD Get_As_String : I_Map
VAR_INPUT
	Key : ANY; // Key used to identify stored value
	sValue : REFERENCE TO STRING; // Variable to store returned item.
END_VAR
VAR_OUTPUT
	bSuccess : BOOL;
END_VAR
END_METHOD

// Gets the value in its generic form associated with the specified key in its generic form without removing it from the map.
// (** Use carefully as this contains the pointer of the actual value in the collection. **)
// If you wish to use this it is recommeded you create a copy of the returned value using MEMCPY
METHOD Get_Generic : I_Map
VAR_INPUT
	Key : T_Generic; // Key used to identify stored value
END_VAR
VAR_OUTPUT
	Value : T_Generic; // Variable to store requested data 
	bSuccess : BOOL;
END_VAR
END_METHOD

// Gets an immutable list of the keys.
METHOD Get_Keys : I_Immutable_List
VAR_INPUT
END_VAR
END_METHOD

// Gets an immutable list of the values.
METHOD Get_Values : I_Immutable_List
VAR_INPUT
END_VAR
END_METHOD

// Insert an element with the provided key and value to the map.
METHOD Insert : I_Map
VAR_INPUT
	Key : ANY; // Key used to identify stored value
	Value : ANY; // Value to store in map with key
END_VAR
VAR_OUTPUT
	bSuccess : BOOL;
END_VAR
END_METHOD

// Insert an element with the provided key and value in their generic forms to the map.
METHOD Insert_Generic : I_Map
VAR_INPUT
	Key : T_Generic; // Key used to identify stored value
	Value : T_Generic; // Value to store in map with key
	bUpdate : BOOL; // If this is true the value will be updated if the key already exists.
END_VAR
VAR_OUTPUT
	bSuccess : BOOL;
END_VAR
END_METHOD

// Removes value with the specified key from the map.
METHOD Remove : I_Map
VAR_INPUT
	Key : ANY; // Key used to identify stored value
END_VAR
VAR_OUTPUT
	bSuccess : BOOL;
END_VAR
END_METHOD

// Removes value with the specified key in its generic form from the map.
METHOD Remove_Generic : I_Map
VAR_INPUT
	Key : T_Generic; // Key used to identify stored value
END_VAR
VAR_OUTPUT
	bSuccess : BOOL;
END_VAR
END_METHOD

// Updates the value at the provided key with the new value in the map.
METHOD Update : I_Map
VAR_INPUT
	Key 	: ANY; // Key used to identify stored value
	Value 	: ANY; // Value to store in map with key
END_VAR
VAR_OUTPUT
	bSuccess : BOOL;
END_VAR
END_METHOD

// Updates the value at the provided key with the new value in their generic forms in the map.
METHOD Update_Generic : I_Map
VAR_INPUT
	Key 	: T_Generic; // Key used to identify stored value
	Value 	: T_Generic; // Value to store in map with key
END_VAR
VAR_OUTPUT
	bSuccess : BOOL;
END_VAR
END_METHOD

// Updates a value in the map for a given key. If the key doesnt exist, it will be inserted.
METHOD Upsert : I_Map
VAR_INPUT
	Key 	: ANY; // Key used to identify stored value
	Value 	: ANY; // Value to store in map with key
END_VAR
VAR_OUTPUT
	bSuccess : BOOL;
END_VAR
END_METHOD

END_INTERFACE

// ITFs/Collections/I_Hash_Set
// Interface for a set implemented using a hash table.
INTERFACE I_Hash_Set EXTENDS I_Set

// Number of buckets in the hash set.
PROPERTY _Bucket_Count : T_Capacity;
GET
END_GET
END_PROPERTY

// Sets the number of buckets in the hash set.
// Existing items are rehashed and redistributed into the new buckets.
METHOD Resize : I_Hash_Set
VAR_INPUT
	Count : T_Capacity;
END_VAR
VAR_OUTPUT
	bSuccess : BOOL;
END_VAR
END_METHOD

END_INTERFACE

// ITFs/Collections/I_Set
// Interface for a set collection.
INTERFACE I_Set EXTENDS I_Collection

// Empties/Clears/Deletes every item in the set.
METHOD Clear : I_Set
END_METHOD

// Checks if item is contained in set.
METHOD Contains : BOOL
VAR_INPUT
	Item : ANY; // Item to find.
END_VAR
END_METHOD

// Gets an immutable list of the values in the set.
METHOD Get_Values : I_Immutable_List
END_METHOD

// Insert item into set.
METHOD Insert 	: I_Set
VAR_INPUT
	Item : ANY; // Data to insert
END_VAR
VAR_OUTPUT
	bSuccess : BOOL; // Indicates whether operation was successful. Success = TRUE, Failure = FALSE
END_VAR
END_METHOD

// Adds new generic item at into set.
// The set will store a copy of the generic item so as to not modify the original value outside it's scope.
METHOD Insert_Generic : I_Set
VAR_INPUT
	Item : T_Generic; // Item to store
END_VAR
VAR_OUTPUT
	bSuccess 	: BOOL; // Indicates whether operation was successful. Success = TRUE, Failure = FALSE
END_VAR
END_METHOD

// Removes item from the set.
METHOD Remove : I_Set
VAR_INPUT
	Item : ANY; // Data to remove
END_VAR
VAR_OUTPUT
	bSuccess : BOOL; // Indicates whether operation was successful. Success = TRUE, Failure = FALSE
END_VAR
END_METHOD

// Removes generic item from the set.
METHOD Remove_Generic : I_Set
VAR_INPUT
	Item : T_Generic; // Data to remove
END_VAR
VAR_OUTPUT
	bSuccess : BOOL; // Indicates whether operation was successful. Success = TRUE, Failure = FALSE
END_VAR
END_METHOD

END_INTERFACE

// ITFs/Collections/I_Queue
// Interface for a queue
INTERFACE I_Queue EXTENDS I_Collection

// Gets an immutable list of the items in the queue.
PROPERTY _Values : I_Immutable_List
GET
END_GET
END_PROPERTY

// Empties/Clears/Deletes every item in the queue.
METHOD Clear : I_Queue
END_METHOD

// Removes item at the front the queue.
METHOD Dequeue : I_Queue
VAR_OUTPUT
	bSuccess : BOOL;
END_VAR
END_METHOD

// Adds item at the back of the queue.
METHOD Enqueue : I_Queue
VAR_INPUT
	Item : ANY; // Item to store.
END_VAR
VAR_OUTPUT
	bSuccess : BOOL;
END_VAR
END_METHOD

// Adds item at the front of the queue.
METHOD Enqueue_At_Front : I_Queue
VAR_INPUT
	Item : ANY; // Item to store.
END_VAR
VAR_OUTPUT
	bSuccess : BOOL;
END_VAR
END_METHOD

// Adds a generic item at the back of the queue.
METHOD Enqueue_Generic : I_Queue
VAR_INPUT
	Item : T_Generic; // Item to store.
	bAt_Front : BOOL; // Enqueues at front if set to TRUE.
END_VAR
VAR_OUTPUT
	bSuccess : BOOL;
END_VAR
END_METHOD

// Gets the item at the front of the queue.
METHOD Get : I_Queue
VAR_INPUT
	Item : ANY; // Variable to store returned item value
END_VAR
VAR_OUTPUT
	bSuccess : BOOL;
END_VAR
END_METHOD

// Gets the item at the front of the queue as a generic.
METHOD Get_Generic : I_Queue
VAR_OUTPUT
	Item : T_Generic; // Variable to store returned item value
	bSuccess : BOOL;
END_VAR
END_METHOD

// Reverses the order of the items in the queue.
METHOD Reverse : I_Queue
VAR_OUTPUT
	bSuccess : BOOL;
END_VAR
END_METHOD

END_INTERFACE

// ITFs/Collections/I_Stack
INTERFACE I_Stack EXTENDS I_Collection

// Gets an immutable list of the items in the stack.
PROPERTY _Values : I_Immutable_List
GET
END_GET
END_PROPERTY

// Empties/Clears/Deletes every item in the stack.
METHOD Clear : I_Stack
END_METHOD

// Gets item at the top of the stack.
METHOD Get : I_Stack
VAR_INPUT
	Item : ANY; // Variable to store returned item value. 
END_VAR
VAR_OUTPUT
	bSuccess : BOOL;
END_VAR
END_METHOD

// Gets item at the top of the stack as a generic.
METHOD Get_Generic : I_Stack
VAR_OUTPUT
	Item : T_Generic; // Variable to store returned item value
	bSuccess : BOOL;
END_VAR
END_METHOD

// Removes item at the top of the stack without returning anything.
METHOD Pop : I_Stack
VAR_OUTPUT
	bSuccess : BOOL;
END_VAR
END_METHOD

// Add item to the top of the stack.
METHOD Push : I_Stack
VAR_INPUT
	Item : ANY; // Item to store.
END_VAR
VAR_OUTPUT
	bSuccess : BOOL;
END_VAR
END_METHOD

// Add generic item to the top of the stack.
METHOD Push_Generic : I_Stack
VAR_INPUT
	Item : T_Generic; // Item to store.
END_VAR
VAR_OUTPUT
	bSuccess : BOOL;
END_VAR
END_METHOD

// Reverses order of items on stack.
METHOD Reverse : I_Stack
VAR_OUTPUT
	bSuccess : BOOL;
END_VAR
END_METHOD

END_INTERFACE

// ITFs/Collections/I_Tree_Map
INTERFACE I_Tree_Map EXTENDS I_Map

// Traversal method for retrieving keys and values in the tree map set.
PROPERTY _Traversal : T_BST_Traversal
GET
END_GET
SET
END_SET
END_PROPERTY

END_INTERFACE

// ITFs/Collections/I_Tree_Set
// Interface for a set implemented using a binary search tree.
INTERFACE I_Tree_Set EXTENDS I_Set

// Traversal method for retrieving values in the tree set.
PROPERTY _Traversal : T_BST_Traversal
GET
END_GET
SET
END_SET
END_PROPERTY

END_INTERFACE

// ITFs/Enumerators/I_Enumerable
INTERFACE I_Enumerable EXTENDS __SYSTEM.IQueryInterface

// Gets an enumerator that iterates through a collection. Returns TRUE if successful.
METHOD Get_Enumerator : BOOL;
VAR_INPUT
	ipEnumerator : REFERENCE TO I_Enumerator;
END_VAR
END_METHOD

END_INTERFACE

// ITFs/Enumerators/I_Enumerator
INTERFACE I_Enumerator EXTENDS __SYSTEM.IQueryInterface

// Gets an item in the collection at current positon of the enumerator.
METHOD Current : I_Enumerator
VAR_INPUT
	Item : ANY;
END_VAR
END_METHOD

// Gets an item in the collection at current positon of the enumerator as a string.
METHOD Current_As_String : I_Enumerable
VAR_INPUT
	sItem : REFERENCE TO STRING;
END_VAR
END_METHOD

// Releases resources allocated to the enumerator. Returns TRUE if successful.
METHOD Dispose : BOOL
VAR_INPUT
END_VAR
END_METHOD

// Advances the enumerator to the next item of the collection.
METHOD Next : BOOL
VAR_INPUT
END_VAR
END_METHOD

// Sets the enumerator to its initial position, which is before the first element in the collection.
METHOD Reset : I_Enumerator
END_METHOD

END_INTERFACE

// ITFs/Iterable/I_Iterable
// Interface that defines the standard structure for indexable collections
INTERFACE I_Iterable EXTENDS __SYSTEM.IQueryInterface

// Index of the first element.
PROPERTY _Begin : T_Position
GET
END_GET
END_PROPERTY

// Index of the last element.
PROPERTY _End : T_Position
GET
END_GET
END_PROPERTY

END_INTERFACE

// ITFs/Misc/I_Copyable
// Interface to apply a copyable attribute to a collection.
INTERFACE I_Copyable EXTENDS __SYSTEM.IQueryInterface

// Copies item in current collection to another collection.
METHOD Copy_To : I_Copyable
VAR_INPUT
	ipCollection : I_Collection;
END_VAR
VAR_OUTPUT
	bSuccess : BOOL;
END_VAR
END_METHOD

END_INTERFACE

// POUs/Function Blocks/Collections/Immutable/FB_Immutable_Array
// Collection that exposes only immutable methods and properties of a collection that implements I_Array.
{attribute 'enable_dynamic_creation'}
FUNCTION_BLOCK FB_Immutable_Array IMPLEMENTS I_Immutable_Array, I_Iterable
VAR_INPUT
	ipArray : I_Array;
END_VAR
VAR
END_VAR

// Index of the first element.
PROPERTY _Begin : T_Position
GET
_Begin := 0;
END_GET
END_PROPERTY

// Number of items in the collection.
PROPERTY _Count : T_Capacity
GET
IF THIS^.ipArray = 0 THEN RETURN; END_IF
_Count := THIS^.ipArray._Count;
END_GET
END_PROPERTY

// Checks if collection is empty.
PROPERTY _Empty : BOOL
GET
IF THIS^.ipArray = 0 THEN _Empty := TRUE; RETURN; END_IF
_Empty := THIS^.ipArray._Empty;
END_GET
END_PROPERTY

// Index of the last element.
PROPERTY _End : T_Position
GET
_End := TO_DINT(THIS^._Count) - 1;
END_GET
END_PROPERTY

// Error status of the collection.
PROPERTY _Error_Status : T_Error
GET
IF THIS^.ipArray = 0 THEN 
	_Error_Status := GVL_Errors.ERR_INVALID_INTERFACE;
	RETURN; 
	END_IF
_Error_Status := THIS^.ipArray._Error_Status;
END_GET
END_PROPERTY

// Checks if item is contained in list.
METHOD Contains : BOOL
VAR_INPUT
	Item : ANY; // Item to find in list
END_VAR
IF THIS^.ipArray = 0 THEN RETURN; END_IF

Contains := THIS^.ipArray.Contains(Item);
END_METHOD

// Gets item from array at specified location without removing it.
METHOD Get : I_Immutable_Array
VAR_INPUT
	Index : T_Position; // Location of item
	Item : ANY;  // Variable to store returned item
END_VAR
VAR_OUTPUT
	bSuccess : BOOL;
END_VAR
Get := THIS^;

IF THIS^.ipArray = 0 THEN RETURN; END_IF

THIS^.ipArray.Get(Index, Item, bSuccess => bSuccess);
END_METHOD

// Returns item as a string, if type to string conversion is supported.
METHOD Get_As_String : I_Immutable_Array
VAR_INPUT
	Index : T_Position; // Location of item
	sItem : REFERENCE TO STRING; // Variable to store returned item.
END_VAR
VAR_OUTPUT
	bSuccess : BOOL;
END_VAR
Get_As_String := THIS^;

IF THIS^.ipArray = 0 THEN RETURN; END_IF

THIS^.ipArray.Get_As_String(Index, sItem, bSuccess => bSuccess);
END_METHOD

// Gets the type of the item at specified location.
METHOD Get_Type_At : I_Immutable_Array
VAR_INPUT
	Index : T_Position;
END_VAR
VAR_OUTPUT
	Item_Type : T_Type := T_Type.TYPE_NONE;
	bSuccess : BOOL;
END_VAR
Get_Type_At := THIS^;

IF THIS^.ipArray = 0 THEN RETURN; END_IF

THIS^.ipArray.Get_Type_At(Index, Item_Type => Item_Type, bSuccess => bSuccess);
END_METHOD

// Find the location of an item in list.
METHOD Search : I_Immutable_Array
VAR_INPUT
	Item : ANY; // Item to find in list
END_VAR
VAR_OUTPUT
	Index : T_Position := -1; //Location of item in list 
	bSuccess : BOOL;
END_VAR
Search := THIS^;

IF THIS^.ipArray = 0 THEN RETURN; END_IF

THIS^.ipArray.Search(Item, Index => Index, bSuccess => bSuccess);
END_METHOD

END_FUNCTION_BLOCK

// POUs/Function Blocks/Collections/Immutable/FB_Immutable_List
// Collection that exposes only immutable methods and properties of a collection that implements I_List.
{attribute 'enable_dynamic_creation'}
FUNCTION_BLOCK FB_Immutable_List IMPLEMENTS I_Immutable_List, I_Iterable
VAR_INPUT
	ipList : I_List;
END_VAR
VAR
END_VAR

// Index of the first element.
PROPERTY _Begin : T_Position
GET
_Begin := 0;
END_GET
END_PROPERTY

// Number of items in the collection.
PROPERTY _Count : T_Capacity
GET
IF THIS^.ipList = 0 THEN RETURN; END_IF

_Count := THIS^.ipList._Count;
END_GET
END_PROPERTY

// Checks if collection is empty.
PROPERTY _Empty : BOOL
GET
IF THIS^.ipList = 0 THEN _Empty := TRUE; RETURN; END_IF
	
_Empty := THIS^.ipList._Empty;
END_GET
END_PROPERTY

// Index of the last element.
PROPERTY _End : T_Position
GET
_End := TO_DINT(THIS^._Count) - 1;
END_GET
END_PROPERTY

// Error status of the collection.
PROPERTY _Error_Status : T_Error
GET
IF THIS^.ipList = 0 THEN 
	_Error_Status := GVL_Errors.ERR_INVALID_INTERFACE;
	RETURN; 
	END_IF
	
_Error_Status := THIS^.ipList._Error_Status;
END_GET
END_PROPERTY

// Checks if item is contained in list.
METHOD Contains : BOOL
VAR_INPUT
	Item : ANY; // Item to find in list
END_VAR
IF THIS^.ipList = 0 THEN RETURN; END_IF

Contains := THIS^.ipList.Contains(Item);
END_METHOD

// Gets item from list at specified location without removing it.
METHOD Get : I_Immutable_List
VAR_INPUT
	Index : T_Position; // Location of item
	Item : ANY;  // Variable to store returned item
END_VAR
VAR_OUTPUT
	bSuccess : BOOL;
END_VAR
Get := THIS^;

IF THIS^.ipList = 0 THEN RETURN; END_IF

THIS^.ipList.Get(Index, Item, bSuccess => bSuccess);
END_METHOD

// Returns item as a string, if type to string conversion is supported.
METHOD Get_As_String : I_Immutable_List
VAR_INPUT
	Index : T_Position; // Location of item
	sItem : REFERENCE TO STRING; // Variable to store returned item.
END_VAR
VAR_OUTPUT
	bSuccess : BOOL;
END_VAR
Get_As_String := THIS^;

IF THIS^.ipList = 0 THEN RETURN; END_IF

THIS^.ipList.Get_As_String(Index, sItem, bSuccess => bSuccess);
END_METHOD

// Gets the type of the item at specified location.
METHOD Get_Type_At : I_Immutable_List
VAR_INPUT
	Index : T_Position;
END_VAR
VAR_OUTPUT
	Item_Type : T_Type := T_Type.TYPE_NONE;
	bSuccess : BOOL;
END_VAR
Get_Type_At := THIS^;

IF THIS^.ipList = 0 THEN RETURN; END_IF

THIS^.ipList.Get_Type_At(Index, Item_Type => Item_Type, bSuccess => bSuccess);
END_METHOD

// Find the location of an item in list.
METHOD Search : I_Immutable_List
VAR_INPUT
	Item : ANY; // Item to find in list
END_VAR
VAR_OUTPUT
	Index : T_Position := -1; //Location of item in list 
	bSuccess : BOOL;
END_VAR
Search := THIS^;

IF THIS^.ipList = 0 THEN RETURN; END_IF

THIS^.ipList.Search(Item, Index => Index, bSuccess => bSuccess);
END_METHOD

END_FUNCTION_BLOCK

// POUs/Function Blocks/Collections/Immutable/FB_Immutable_Map
// Collection that exposes only immutable methods and properties of a collection that implements I_Map.
{attribute 'enable_dynamic_creation'}
FUNCTION_BLOCK FB_Immutable_Map IMPLEMENTS I_Immutable_Map
VAR_INPUT
	ipMap : I_Map;
END_VAR
VAR_STAT
	fbDefault_Immutable_List : FB_Immutable_List;
END_VAR

// Number of items in the collection.
PROPERTY _Count : T_Capacity
GET
IF THIS^.ipMap = 0 THEN RETURN; END_IF
	
_Count := THIS^.ipMap._Count;
END_GET
END_PROPERTY

// Checks if collection is empty.
PROPERTY _Empty : BOOL
GET
IF THIS^.ipMap = 0 THEN _Empty := TRUE; RETURN; END_IF
	
_Empty := THIS^.ipMap._Empty;
END_GET
END_PROPERTY

// Error status of the collection.
PROPERTY _Error_Status : T_Error
GET
IF THIS^.ipMap = 0 THEN 
	_Error_Status := GVL_Errors.ERR_INVALID_INTERFACE;
	RETURN; 
	END_IF
	
_Error_Status := THIS^.ipMap._Error_Status;
END_GET
END_PROPERTY

// Checks if key is contained in the map.
METHOD Contains : BOOL
VAR_INPUT
	Key : ANY; // Key to find.
END_VAR
IF THIS^.ipMap = 0 THEN RETURN; END_IF

Contains := THIS^.ipMap.Contains(Key);
END_METHOD

// Gets the value associated with the specified key without removing it from the map.
METHOD Get : I_Immutable_Map
VAR_INPUT
	Key : ANY; // Key used to identify stored value
	Value : ANY; // Variable to store requested data 
END_VAR
VAR_OUTPUT
	bSuccess : BOOL;
END_VAR
Get := THIS^;

IF THIS^.ipMap = 0 THEN RETURN; END_IF

THIS^.ipMap.Get(Key, Value, bSuccess => bSuccess);
END_METHOD

// Returns value as a string, if type to string conversion is supported.
METHOD Get_As_String : I_Immutable_Map
VAR_INPUT
	Key : ANY; // Key used to identify stored value
	sValue : REFERENCE TO STRING; // Variable to store returned item.
END_VAR
VAR_OUTPUT
	bSuccess : BOOL;
END_VAR
Get_As_String := THIS^;

IF THIS^.ipMap = 0 THEN RETURN; END_IF

THIS^.ipMap.Get_As_String(Key, sValue, bSuccess => bSuccess);
END_METHOD

// Gets an immutable list of the keys.
METHOD Get_Keys : I_Immutable_List
VAR
END_VAR
IF THIS^.ipMap = 0 THEN 
	Get_Keys := THIS^.fbDefault_Immutable_List;
	RETURN; 
	END_IF

Get_Keys := THIS^.ipMap.Get_Values();
END_METHOD

// Gets an immutable list of the values in the map.
METHOD Get_Values : I_Immutable_List
IF THIS^.ipMap = 0 THEN 
	Get_Values := THIS^.fbDefault_Immutable_List;
	RETURN; 
	END_IF

Get_Values := THIS^.ipMap.Get_Values();
END_METHOD

END_FUNCTION_BLOCK

// POUs/Function Blocks/Collections/Immutable/FB_Immutable_Set
// Collection that exposes only immutable methods and properties of a collection that implements I_Set.
{attribute 'enable_dynamic_creation'}
FUNCTION_BLOCK FB_Immutable_Set IMPLEMENTS I_Immutable_Set
VAR_INPUT
	ipSet : I_Set;
END_VAR
VAR_STAT
	fbDefault_Immutable_List : FB_Immutable_List;
END_VAR

// Number of items in the collection.
PROPERTY _Count : T_Capacity
GET
IF THIS^.ipSet = 0 THEN RETURN; END_IF
	
_Count := THIS^.ipSet._Count;
END_GET
END_PROPERTY

// Checks if collection is empty.
PROPERTY _Empty : BOOL
GET
IF THIS^.ipSet = 0 THEN _Empty := TRUE; RETURN; END_IF
	
_Empty := THIS^.ipSet._Empty;
END_GET
END_PROPERTY

// Error status of the collection.
PROPERTY _Error_Status : T_Error
GET
IF THIS^.ipSet = 0 THEN 
	_Error_Status := GVL_Errors.ERR_INVALID_INTERFACE;
	RETURN; 
	END_IF
	
_Error_Status := THIS^.ipSet._Error_Status;
END_GET
END_PROPERTY

// Checks if item is contained in set.
METHOD Contains : BOOL
VAR_INPUT
	Item : ANY; // Item to find.
END_VAR
IF THIS^.ipSet = 0 THEN RETURN; END_IF

Contains := THIS^.ipSet.Contains(Item);
END_METHOD

// Gets an immutable list of the values in the set.
METHOD Get_Values : I_Immutable_List
VAR
END_VAR
IF THIS^.ipSet = 0 THEN 
	Get_Values := THIS^.fbDefault_Immutable_List;
	RETURN; 
	END_IF

Get_Values := THIS^.ipSet.Get_Values();
END_METHOD

END_FUNCTION_BLOCK

// POUs/Function Blocks/Collections/FB_Array
// Static array function block.
{attribute 'enable_dynamic_creation'}
{attribute 'no_assign'}
{attribute 'no_explicit_call' := 'direct call for this function block is not allowed'}
FUNCTION_BLOCK FB_Array EXTENDS FB_Collection IMPLEMENTS I_Array, I_Iterable //, I_Enumerable, I_Copyable
VAR
	pBuffer : POINTER TO T_Generic;
END_VAR

// Index of the first element.
PROPERTY _Begin : T_Position
GET
_Begin := 0;
END_GET
END_PROPERTY

// Index of the last element.
PROPERTY _End : T_Position
GET
_End := TO_DINT(THIS^._Count) - 1;
END_GET
END_PROPERTY

// Checks if item is contained in array.
METHOD Contains : BOOL
VAR_INPUT
	Item : ANY; // Item to find.
END_VAR
THIS^.Search(Item, bSuccess => Contains);
END_METHOD

{attribute 'hide'}
METHOD FB_exit : BOOL
VAR_INPUT
	bInCopyCode : BOOL; // if TRUE, the exit method is called for exiting an instance that is copied afterwards (online change).
END_VAR
VAR
	i : T_Capacity;
END_VAR
// Return if it's an online change.
IF bInCopyCode THEN RETURN; END_IF

THIS^.Clear_Error();

IF THIS^.pBuffer = 0 THEN THIS^._Count := 0; RETURN; END_IF

FOR i := 0 TO THIS^._Count - 1 DO
	F_Delete_Generic(THIS^.pBuffer[i]);
	END_FOR
	
THIS^._Count := 0;	
__DELETE(THIS^.pBuffer);
END_METHOD

{attribute 'hide'}
METHOD FB_init : BOOL
VAR_INPUT
	bInitRetains 	: BOOL; // if TRUE, the retain variables are initialized (warm start / cold start)
	bInCopyCode 	: BOOL; // if TRUE, the instance afterwards gets moved into the copy code (online change)
	Count 			: T_Capacity; // The size of the array.
END_VAR
VAR
	i : T_Capacity;
END_VAR
// Return if it's an online change.
IF bInCopyCode THEN RETURN; END_IF

THIS^._Count := Count;

IF Count = 0 THEN RETURN; END_IF

THIS^.pBuffer := F_Malloc_Generic(Count, Error => THIS^.Error);
END_METHOD

// Gets item from array at specified location.
METHOD Get : I_Array
VAR_INPUT
	Index : T_Position; // Location of item.
	Item : ANY;  // Variable to store returned item.
END_VAR
VAR_OUTPUT
	bSuccess : BOOL;
END_VAR
Get := THIS^;

IF THIS^.pBuffer = 0 THEN THIS^._Error_Status := GVL_Errors.ERR_MALLOC_FAILED; RETURN; END_IF

IF Index < 0 OR_ELSE Index >= THIS^._Count THEN THIS^._Error_Status := GVL_Errors.ERR_INDEX_OUT_OF_BOUNDS; RETURN; END_IF

IF NOT F_Matching_Generics(Item, THIS^.pBuffer[Index]) THEN THIS^._Error_Status := GVL_Errors.ERR_TYPE_MISMATCH; RETURN; END_IF
	
F_Copy_Generic_Value(THIS^.pBuffer[Index], Item);
bSuccess := TRUE;
THIS^.Clear_Error();
END_METHOD

// Returns item as a string, if type to string conversion is supported.
METHOD Get_As_String : I_Array
VAR_INPUT
	Index : T_Position; // Location of item.
	sItem : REFERENCE TO STRING; // Variable to store returned item.
END_VAR
VAR_OUTPUT
	bSuccess : BOOL;
END_VAR
Get_As_String := THIS^;

IF THIS^.pBuffer = 0 THEN 
	THIS^._Error_Status := GVL_Errors.ERR_MALLOC_FAILED; 
	RETURN; 
	END_IF

IF NOT __ISVALIDREF(sItem) THEN 
	THIS^._Error_Status := GVL_Errors.ERR_INVALID_REFERENCE;
	RETURN;
	END_IF

IF Index < 0 OR_ELSE Index >= THIS^._Count THEN 
	THIS^._Error_Status := GVL_Errors.ERR_INDEX_OUT_OF_BOUNDS;
	RETURN; 
	END_IF
	
CASE THIS^.pBuffer[Index].TypeClass OF
	T_Type.TYPE_STRING:
		Tc2_Utilities.STRNCPY(ADR(sItem), THIS^.pBuffer[Index].pValue, MIN(Tc2_Utilities.LEN2(ADR(sItem))+1, TO_UDINT(THIS^.pBuffer[Index].diSize)));
		THIS^.Clear_Error();

	T_Type.TYPE_WSTRING:
		Tc2_Utilities.WSTRING_TO_STRING2(ADR(sItem), THIS^.pBuffer[Index].pValue, MIN(Tc2_Utilities.LEN2(ADR(sItem))+1, TO_UDINT(THIS^.pBuffer[Index].diSize)));
		THIS^.Clear_Error();
ELSE
	sItem := F_Generic_To_String(THIS^.pBuffer[Index], bSuccess => bSuccess, Error => THIS^.Error);
	END_CASE
END_METHOD

// Gets an item from the array in it's generic form.
// (** Use carefully as this contains the pointer of the actual value in the collection. **)
// If you wish to use this it is recommeded you create a copy of the returned value using MEMMOVE or MEMCPY
METHOD Get_Generic : I_Array
VAR_INPUT
	Index : T_Position; // Location of item.
END_VAR
VAR_OUTPUT
	Item : T_Generic;
	bSuccess : BOOL;
END_VAR
Get_Generic := THIS^;

IF THIS^.pBuffer = 0 THEN THIS^._Error_Status := GVL_Errors.ERR_MALLOC_FAILED; RETURN; END_IF

IF Index < 0 OR_ELSE Index >= THIS^._Count THEN THIS^._Error_Status := GVL_Errors.ERR_INDEX_OUT_OF_BOUNDS; RETURN; END_IF

Item := THIS^.pBuffer[Index];
bSuccess := TRUE;
THIS^.Clear_Error();
END_METHOD

// Gets the type of the item at specified location.
METHOD Get_Type_At : I_Array
VAR_INPUT
	Index : T_Position;
END_VAR
VAR_OUTPUT
	Item_Type : T_Type := T_Type.TYPE_NONE;
	bSuccess : BOOL;
END_VAR
VAR
	Tmp : T_Generic;
END_VAR
Get_Type_At := THIS^;

THIS^.Get_Generic(Index, Item => Tmp, bSuccess => bSuccess);

IF bSuccess THEN Item_Type := Tmp.TypeClass; END_IF
END_METHOD

// Reverses the order of items in the array.
METHOD Reverse : I_Array
VAR_OUTPUT
	bSuccess : BOOL;
END_VAR
VAR
	i : T_Capacity;
END_VAR
Reverse := THIS^;

IF THIS^.pBuffer = 0 THEN THIS^._Error_Status := GVL_Errors.ERR_MALLOC_FAILED; RETURN; END_IF

IF NOT THIS^._Empty THEN
	FOR i := 0 TO (THIS^._Count/2) - 1 DO
		F_Swap_Generics(THIS^.pBuffer[i], THIS^.pBuffer[THIS^._Count - i - 1]);
		END_FOR
	END_IF

bSuccess := TRUE;
THIS^.Clear_Error();
END_METHOD

// Find the location of an item in the array.
METHOD Search : I_Array
VAR_INPUT
	Item : ANY; // Item to find.
END_VAR
VAR_OUTPUT
	Index : T_Position; //Location of item.
	bSuccess : BOOL;
END_VAR
VAR
	i : T_Position;
END_VAR
Search := THIS^;

IF THIS^.pBuffer = 0 THEN THIS^._Error_Status := GVL_Errors.ERR_MALLOC_FAILED; RETURN; END_IF

FOR i := 0 TO THIS^._Count - 1 DO
	CASE F_Compare_Generics(Item, THIS^.pBuffer[i]) OF
		T_Comparison.Equal:
			bSuccess := TRUE;
			THIS^.Clear_Error();
			Index := i;
			RETURN;
		END_CASE
	END_FOR
END_METHOD

// Changes the item at the specified location in the array.
METHOD Set : I_Array
VAR_INPUT
	Index 	: T_Position; // Location of item.
	Item 	: ANY; 	// Item to store.
END_VAR
VAR_OUTPUT
	bSuccess : BOOL;
END_VAR
Set := THIS^;

THIS^.Set_Generic(Index, Item, bSuccess => bSuccess);
END_METHOD

// Changes the item at the specified location in the array in it's generic form.
METHOD Set_Generic : I_Array
VAR_INPUT
	Index : T_Position; // Location of item.
	Item : T_Generic; // Item to store.
END_VAR
VAR_OUTPUT
	bSuccess : BOOL;
END_VAR
VAR
	Tmp : T_Generic;
END_VAR
Set_Generic := THIS^;

IF THIS^.pBuffer = 0 THEN THIS^._Error_Status := GVL_Errors.ERR_MALLOC_FAILED; RETURN; END_IF

IF Index < 0 OR_ELSE Index >= THIS^._Count THEN THIS^._Error_Status :=  GVL_Errors.ERR_INDEX_OUT_OF_BOUNDS; RETURN; END_IF

Tmp := F_Clone_Generic(Item, bSuccess => bSuccess, Error => THIS^.Error);

IF NOT bSuccess THEN THIS^._Error_Status := GVL_Errors.ERR_MALLOC_FAILED; RETURN; END_IF

F_Delete_Generic(THIS^.pBuffer[Index]);

THIS^.pBuffer[Index] := Tmp;
END_METHOD

// Swaps item at index with item at index B.
METHOD Swap : I_Array
VAR_INPUT
	Index_A, Index_B : T_Position;
END_VAR
VAR_OUTPUT
	bSuccess : BOOL;
END_VAR
Swap := THIS^;

IF THIS^.pBuffer = 0 THEN THIS^._Error_Status := GVL_Errors.ERR_MALLOC_FAILED; RETURN; END_IF

IF Index_A < 0 OR_ELSE Index_A >= THIS^._Count OR_ELSE Index_B < 0 OR_ELSE Index_B >= THIS^._Count THEN
	THIS^._Error_Status := GVL_Errors.ERR_INDEX_OUT_OF_BOUNDS;
	RETURN;
	END_IF
	
F_Swap_Generics(THIS^.pBuffer[Index_A], THIS^.pBuffer[Index_B], bSuccess => bSuccess, Error => THIS^.Error);
END_METHOD

END_FUNCTION_BLOCK

// POUs/Function Blocks/Collections/FB_Collection
// Abstract class/Function Block that all collections inherit.
// Contains inheritable helper methods and base implementation
// for methods and properties for creating a collection.
{attribute 'enable_dynamic_creation'}
{attribute 'no_explicit_call' := 'direct call for this function block is not allowed'}
FUNCTION_BLOCK ABSTRACT FB_Collection IMPLEMENTS I_Collection
VAR
	Count : T_Capacity;
	Error : T_Error := GVL_Errors.ERR_NO_ERROR;
END_VAR

METHOD PROTECTED Clear_Error
VAR_INPUT
END_VAR
THIS^._Error_Status := F_Error(0,0,'');
END_METHOD

// Decrement collection count by 1.
METHOD PROTECTED Decrement_Count
THIS^._Count := THIS^._Count - 1;
END_METHOD

// Increments collection count by 1
METHOD PROTECTED Increment_Count
VAR_INPUT
END_VAR
THIS^._Count := THIS^._Count + 1;
END_METHOD

// Number of items in the collection.
PROPERTY _Count : T_Capacity
GET
_Count := THIS^.Count;
END_GET
SET
PROTECTED 
VAR
END_VAR
THIS^.Count := _Count;
END_SET
END_PROPERTY

// Checks if collection is empty.
PROPERTY _Empty : BOOL
GET
_Empty := THIS^._Count <= 0;
END_GET
END_PROPERTY

// Error status of the collection.
PROPERTY _Error_Status : T_Error
GET
_Error_Status := THIS^.Error;
END_GET
SET
PROTECTED 
VAR
END_VAR
THIS^.Error := _Error_Status;
END_SET
END_PROPERTY

END_FUNCTION_BLOCK

// POUs/Functions/F_Error
// Error Function: Passes error code and message to type ST_ERROR when bStatus = TRUE.  
FUNCTION F_Error : T_Error
VAR_INPUT
	bStatus : BOOL; 		// Trigger to pass code and message | Note: Default is FALSE
	nCode 	: DINT; 		// Code to pass to error struct | Note: code is 0 if there is no error
	sSource : T_MaxString; 	// Message to pass to error struct | Note: message is 'No Error.'  if there is no error
END_VAR
VAR
	Tmp_Error : T_Error;
END_VAR

Tmp_Error.bSTATUS := bStatus; 
IF bStatus THEN 
	Tmp_Error.nCODE := nCode; 
	Tmp_Error.sSOURCE := sSource;
ELSE 
	Tmp_Error := GVL_Errors.ERR_NO_ERROR; 
	END_IF
	
F_Error := Tmp_Error;

END_FUNCTION

// POUs/Functions/F_Delete_Generic
// Deletes a generic's value.
FUNCTION F_Delete_Generic
VAR_INPUT
	Source : REFERENCE TO T_Generic;
END_VAR
VAR_OUTPUT
	bSuccess : BOOL;
	Error : T_Error := GVL_Errors.ERR_NO_ERROR;
END_VAR

IF (NOT __ISVALIDREF(Source)) THEN 
	Error := GVL_Errors.ERR_INVALID_REFERENCE;
	RETURN;
	END_IF

CASE Tc2_System.F_CheckMemoryArea(Source.pValue, 1) OF
	Tc2_System.E_TcMemoryArea.Dynamic: __DELETE(Source.pValue);
ELSE
	Source.pValue := 0;
	END_CASE

Source.diSize := 0;
Source.TypeClass := T_Type.TYPE_NONE;

bSuccess := TRUE;

END_FUNCTION

// POUs/Functions/F_Malloc_Generic
// Allocates memory for T_Generic.
FUNCTION F_Malloc_Generic : POINTER TO T_Generic
VAR_INPUT
	Count : T_Capacity;
END_VAR
VAR_OUTPUT
	bSuccess : BOOL;
	Error : T_Error := GVL_Errors.ERR_NO_ERROR;
END_VAR
VAR
	i : T_Capacity;
	Size : UDINT;
END_VAR

IF Count = 0 THEN bSuccess := TRUE; RETURN; END_IF

Size := TO_UDINT(SIZEOF(T_Generic) * Count);
F_Malloc_Generic := __NEW(BYTE, Size);

IF F_Malloc_Generic = 0 THEN 
	Error := GVL_Errors.ERR_MALLOC_FAILED;
	RETURN;
	END_IF

FOR i := 0 TO count - 1 DO
	F_Malloc_Generic[i].TypeClass := T_Type.TYPE_NONE;
	END_FOR

bSuccess := TRUE;

END_FUNCTION

// POUs/Functions/F_Matching_Generics
// Checks if 2 generics can be compared to see if they match (same size, same class). Match = TRUE, Not Matching = FALSE.
// The exception is strings. If 2 generics are strings they're considered to be matching regardless of size;
FUNCTION F_Matching_Generics : BOOL
VAR_INPUT
	A, B : T_Generic;
END_VAR

F_Matching_Generics := 
	(A.diSize = B.diSize AND_THEN A.TypeClass = B.TypeClass)
	OR_ELSE
	(A.TypeClass = __SYSTEM.TYPE_CLASS.TYPE_STRING AND_THEN B.TypeClass = __SYSTEM.TYPE_CLASS.TYPE_STRING)
	OR_ELSE
	(A.TypeClass = __SYSTEM.TYPE_CLASS.TYPE_WSTRING AND_THEN B.TypeClass = __SYSTEM.TYPE_CLASS.TYPE_WSTRING);

END_FUNCTION

// POUs/Functions/F_Copy_Generic_Value
// Copies the value of a generic from one location to another.
FUNCTION F_Copy_Generic_Value
VAR_INPUT
	Source, Destination : REFERENCE TO T_Generic;
END_VAR
VAR_OUTPUT
	bSuccess : BOOL;
	Error : T_Error := GVL_Errors.ERR_NO_ERROR;
END_VAR

IF NOT( __ISVALIDREF(Source) OR_ELSE __ISVALIDREF(Destination)) THEN 
	Error := GVL_Errors.ERR_INVALID_REFERENCE;
	RETURN; 
	END_IF

bSuccess := Tc2_System.MEMCPY(
	Destination.pValue, Source.pValue, 
	TO_UDINT(MIN(Source.diSize, Destination.diSize))) > 0;

END_FUNCTION

// POUs/Functions/F_Generic_To_String
FUNCTION F_Generic_To_String : T_MaxString
VAR_INPUT
	 Value : T_Generic;
END_VAR
VAR_OUTPUT
	bSuccess : BOOL;
	Error : T_Error := GVL_Errors.ERR_NO_ERROR;
END_VAR
VAR	
	pBool			: POINTER TO BOOL;
    pByte			: POINTER TO BYTE;
    pWord			: POINTER TO WORD;
    pDWord			: POINTER TO DWORD;
    pLWord			: POINTER TO LWORD;
    pSint			: POINTER TO SINT;
    pInt			: POINTER TO INT;
    pDint			: POINTER TO DINT;
    pLint			: POINTER TO LINT;
    pUSint			: POINTER TO USINT;
    pUInt			: POINTER TO UINT;
    pUDint			: POINTER TO UDINT;
    pULint			: POINTER TO ULINT;
    pReal			: POINTER TO REAL;
    pLReal			: POINTER TO LREAL;
    pString			: POINTER TO STRING(255);
    pWString		: POINTER TO WSTRING;
    pTime			: POINTER TO TIME;
    pDate			: POINTER TO DATE;
    pDate_And_Time	: POINTER TO DATE_AND_TIME;
    pTime_Of_Day	: POINTER TO TIME_OF_DAY;
    pPointer		: PVOID;
	pLTime 			: POINTER TO LTIME;
END_VAR

IF Value.pValue = 0 THEN 
	Error := GVL_Errors.ERR_INVALID_REFERENCE;
	RETURN;
	END_IF;

CASE Value.TypeClass OF 
	__SYSTEM.TYPE_CLASS.TYPE_BOOL:
		pBool := Value.pValue;
		F_Generic_To_String := TO_STRING(pBool^);
		
    __SYSTEM.TYPE_CLASS.TYPE_BYTE:
		pByte := Value.pValue;
		F_Generic_To_String := TO_STRING(pByte^);
		
    __SYSTEM.TYPE_CLASS.TYPE_WORD:
		pWord := Value.pValue;
		F_Generic_To_String := TO_STRING(pWord^);
		
    __SYSTEM.TYPE_CLASS.TYPE_DWORD:
		pDWord := Value.pValue;
		F_Generic_To_String := TO_STRING(pDWord^);
		
    __SYSTEM.TYPE_CLASS.TYPE_LWORD:
		pLWord := Value.pValue;
		F_Generic_To_String := TO_STRING(pLWord^);
		
    __SYSTEM.TYPE_CLASS.TYPE_SINT:
		pSint := Value.pValue;
		F_Generic_To_String := TO_STRING(pSint^);
		
    __SYSTEM.TYPE_CLASS.TYPE_INT:
		pInt := Value.pValue;
		F_Generic_To_String := TO_STRING(pInt^);
		
    __SYSTEM.TYPE_CLASS.TYPE_DINT:
		pDint := Value.pValue;
		F_Generic_To_String := TO_STRING(pDint^);
		
    __SYSTEM.TYPE_CLASS.TYPE_LINT:
		pLint := Value.pValue;
		F_Generic_To_String := TO_STRING(pLint^);
		
    __SYSTEM.TYPE_CLASS.TYPE_USINT:
		pUSint := Value.pValue;
		F_Generic_To_String := TO_STRING(pUSint^);
		
    __SYSTEM.TYPE_CLASS.TYPE_UINT:
		pUInt := Value.pValue;
		F_Generic_To_String := TO_STRING(pUInt^);
		
    __SYSTEM.TYPE_CLASS.TYPE_UDINT:
		pUDint := Value.pValue;
		F_Generic_To_String := TO_STRING(pUDint^);
		
    __SYSTEM.TYPE_CLASS.TYPE_ULINT:
		pULint := Value.pValue;
		F_Generic_To_String := TO_STRING(pULint^);
		
   __SYSTEM.TYPE_CLASS.TYPE_REAL:
		pReal := Value.pValue;
		F_Generic_To_String := TO_STRING(pReal^);
		
    __SYSTEM.TYPE_CLASS.TYPE_LREAL:
		pLReal := Value.pValue;
		F_Generic_To_String := TO_STRING(pLReal^);
		
    __SYSTEM.TYPE_CLASS.TYPE_STRING:
		pString := Value.pValue;
		F_Generic_To_String := TO_STRING(pString^);
		
   __SYSTEM.TYPE_CLASS.TYPE_WSTRING:
		pWString := Value.pValue;
		F_Generic_To_String := TO_STRING(pWString^);
		
    __SYSTEM.TYPE_CLASS.TYPE_TIME:
		pTime := Value.pValue;
		F_Generic_To_String := TO_STRING(pTime^);
		
    __SYSTEM.TYPE_CLASS.TYPE_DATE:
		pDate := Value.pValue;
		F_Generic_To_String := TO_STRING(pDate^);
		
    __SYSTEM.TYPE_CLASS.TYPE_DATEANDTIME:
		pDate_And_Time := Value.pValue;
		F_Generic_To_String := TO_STRING(pDate_And_Time^);
		
    __SYSTEM.TYPE_CLASS.TYPE_TIMEOFDAY:
		pTime_Of_Day := Value.pValue;
		F_Generic_To_String := TO_STRING(pTime_Of_Day^);
	
	__SYSTEM.TYPE_CLASS.TYPE_POINTER:
		F_Generic_To_String := TO_STRING(Value.pValue);
		
	__SYSTEM.TYPE_CLASS.TYPE_LTIME:
		pLTime := Value.pValue;
		F_Generic_To_String := TO_STRING(pLTime^);
ELSE
	Error := GVL_Errors.ERR_INVALID_CONVERSION;
	RETURN;
	END_CASE
	
bSuccess := TRUE;

END_FUNCTION

// POUs/Functions/F_Swap_Generics
// Swaps generic A with B.
FUNCTION F_Swap_Generics
VAR_INPUT
	A, B : REFERENCE TO T_Generic;
END_VAR
VAR_OUTPUT
	bSuccess : BOOL;
	Error : T_Error := GVL_Errors.ERR_NO_ERROR;
END_VAR
VAR
	Tmp : T_Generic;
END_VAR

IF NOT(__ISVALIDREF(A) AND_THEN __ISVALIDREF(B)) THEN 
	Error := GVL_Errors.ERR_INVALID_REFERENCE;
	RETURN;
	END_IF

Tmp := A;
A := B;
B := Tmp;
bSuccess := TRUE;

END_FUNCTION

// POUs/Functions/F_Compare_Generics
// Compares generic value A to generic value B and returns the evaluation.
FUNCTION F_Compare_Generics : T_Comparison
VAR_INPUT
	A, B : T_Generic;
END_VAR
VAR_OUTPUT
	bUndefined : BOOL; // If TRUE, values were compared but truthfulness of comparison cannot be verified. 
END_VAR
VAR
	fA, fB : LREAL;
	tA, tB : LTIME;
	dtA, dtB : DT;
END_VAR

IF F_Is_Numeric_Generic(A) AND_THEN F_Is_Numeric_Generic(B) THEN
	fA := F_Generic_To_LREAL(A);
	fB := F_Generic_To_LREAL(B);
	F_Compare_Generics := SEL(fA = fB, SEL(fA > fB, T_Comparison.Less, T_Comparison.Greater), T_Comparison.Equal);
	RETURN;
	END_IF
	
IF F_Is_Time_Generic(A) AND_THEN F_Is_Time_Generic(B) THEN
	tA := F_Generic_To_LTIME(A);
	tB := F_Generic_To_LTIME(B);
	F_Compare_Generics := SEL(tA = tB, SEL(tA > tB, T_Comparison.Less, T_Comparison.Greater), T_Comparison.Equal);
	RETURN;
	END_IF

IF F_Is_Date_Generic(A) AND_THEN F_Is_Date_Generic(B) THEN
	dtA := F_Generic_To_DT(A);
	dtB := F_Generic_To_DT(B);
	F_Compare_Generics := SEL(dtA = dtB, SEL(dtA > dtB, T_Comparison.Less, T_Comparison.Greater), T_Comparison.Equal);
	RETURN;
	END_IF

IF F_Matching_Generics(A, B) THEN
	bUndefined := A.TypeClass = T_Type.TYPE_USERDEF;
	A.diSize := SEL(A.TypeClass = T_Type.TYPE_STRING, SEL(A.TypeClass = T_Type.TYPE_WSTRING, A.diSize, TO_DINT(Tc2_Utilities.WLEN2(A.pValue))) , TO_DINT(Tc2_Utilities.LEN2(A.pValue)));
	B.diSize := SEL(B.TypeClass = T_Type.TYPE_STRING, SEL(B.TypeClass = T_Type.TYPE_WSTRING, B.diSize, TO_DINT(Tc2_Utilities.WLEN2(B.pValue))) , TO_DINT(Tc2_Utilities.LEN2(B.pValue)));
	CASE Tc2_System.MEMCMP(A.pValue, B.pValue, TO_UDINT(MIN(A.diSize, B.diSize))) OF
		-1		: F_Compare_Generics := T_Comparison.Less;
		0		: F_Compare_Generics := T_Comparison.Equal;
		1		: F_Compare_Generics := T_Comparison.Greater;
		16#FF	:
			bUndefined := TRUE; 
			F_Compare_Generics := SEL(A.diSize = B.diSize, SEL(A.diSize > B.diSize, T_Comparison.Less, T_Comparison.Greater), T_Comparison.Equal);
		END_CASE
	RETURN;
	END_IF
	
bUndefined := TRUE;
F_Compare_Generics := SEL(A.TypeClass > B.TypeClass, T_Comparison.Less, T_Comparison.Greater);

END_FUNCTION

// POUs/Functions/F_Is_Numeric_Generic
// Checks if a generic is numeric.
FUNCTION F_Is_Numeric_Generic : BOOL
VAR_INPUT
	Value : T_Generic;
END_VAR
VAR
END_VAR

CASE Value.TypeClass OF
	__SYSTEM.TYPE_CLASS.TYPE_BOOL,
	__SYSTEM.TYPE_CLASS.TYPE_BYTE,
	__SYSTEM.TYPE_CLASS.TYPE_WORD,
	__SYSTEM.TYPE_CLASS.TYPE_DWORD,
	__SYSTEM.TYPE_CLASS.TYPE_LWORD,
	__SYSTEM.TYPE_CLASS.TYPE_SINT,
	__SYSTEM.TYPE_CLASS.TYPE_INT,
	__SYSTEM.TYPE_CLASS.TYPE_DINT,
	__SYSTEM.TYPE_CLASS.TYPE_LINT,
	__SYSTEM.TYPE_CLASS.TYPE_USINT,
	__SYSTEM.TYPE_CLASS.TYPE_UINT,
	__SYSTEM.TYPE_CLASS.TYPE_UDINT,
	__SYSTEM.TYPE_CLASS.TYPE_ULINT,
	__SYSTEM.TYPE_CLASS.TYPE_REAL,
	__SYSTEM.TYPE_CLASS.TYPE_LREAL,
	__SYSTEM.TYPE_CLASS.TYPE_POINTER:
		F_Is_Numeric_Generic := TRUE;
END_CASE

END_FUNCTION

// POUs/Functions/F_Generic_To_LREAL
FUNCTION F_Generic_To_LREAL : LREAL
VAR_INPUT
	 Value : T_Generic;
END_VAR
VAR_OUTPUT
	bSuccess : BOOL;
	Error : T_Error := GVL_Errors.ERR_NO_ERROR;
END_VAR
VAR	
	pBool			: POINTER TO BOOL;
    pByte			: POINTER TO BYTE;
    pWord			: POINTER TO WORD;
    pDWord			: POINTER TO DWORD;
    pLWord			: POINTER TO LWORD;
    pSint			: POINTER TO SINT;
    pInt			: POINTER TO INT;
    pDint			: POINTER TO DINT;
    pLint			: POINTER TO LINT;
    pUSint			: POINTER TO USINT;
    pUInt			: POINTER TO UINT;
    pUDint			: POINTER TO UDINT;
    pULint			: POINTER TO ULINT;
    pReal			: POINTER TO REAL;
    pLReal			: POINTER TO LREAL;
    pString			: POINTER TO STRING(255);
    pWString		: POINTER TO WSTRING;
    pTime			: POINTER TO TIME;
    pDate			: POINTER TO DATE;
    pDate_And_Time	: POINTER TO DATE_AND_TIME;
    pTime_Of_Day	: POINTER TO TIME_OF_DAY;
    pPointer		: PVOID;
	pLTime 			: POINTER TO LTIME;
END_VAR

IF Value.pValue = 0 THEN 
	Error := GVL_Errors.ERR_INVALID_REFERENCE;
	RETURN;
	END_IF;

CASE Value.TypeClass OF 
	__SYSTEM.TYPE_CLASS.TYPE_BOOL:
		pBool := Value.pValue;
		F_Generic_To_LREAL := TO_LREAL(pBool^);
		
    __SYSTEM.TYPE_CLASS.TYPE_BYTE:
		pByte := Value.pValue;
		F_Generic_To_LREAL := TO_LREAL(pByte^);
		
    __SYSTEM.TYPE_CLASS.TYPE_WORD:
		pWord := Value.pValue;
		F_Generic_To_LREAL := TO_LREAL(pWord^);
		
    __SYSTEM.TYPE_CLASS.TYPE_DWORD:
		pDWord := Value.pValue;
		F_Generic_To_LREAL := TO_LREAL(pDWord^);
		
    __SYSTEM.TYPE_CLASS.TYPE_LWORD:
		pLWord := Value.pValue;
		F_Generic_To_LREAL := TO_LREAL(pLWord^);
		
    __SYSTEM.TYPE_CLASS.TYPE_SINT:
		pSint := Value.pValue;
		F_Generic_To_LREAL := TO_LREAL(pSint^);
		
    __SYSTEM.TYPE_CLASS.TYPE_INT:
		pInt := Value.pValue;
		F_Generic_To_LREAL := TO_LREAL(pInt^);
		
    __SYSTEM.TYPE_CLASS.TYPE_DINT:
		pDint := Value.pValue;
		F_Generic_To_LREAL := TO_LREAL(pDint^);
		
    __SYSTEM.TYPE_CLASS.TYPE_LINT:
		pLint := Value.pValue;
		F_Generic_To_LREAL := TO_LREAL(pLint^);
		
    __SYSTEM.TYPE_CLASS.TYPE_USINT:
		pUSint := Value.pValue;
		F_Generic_To_LREAL := TO_LREAL(pUSint^);
		
    __SYSTEM.TYPE_CLASS.TYPE_UINT:
		pUInt := Value.pValue;
		F_Generic_To_LREAL := TO_LREAL(pUInt^);
		
    __SYSTEM.TYPE_CLASS.TYPE_UDINT:
		pUDint := Value.pValue;
		F_Generic_To_LREAL := TO_LREAL(pUDint^);
		
    __SYSTEM.TYPE_CLASS.TYPE_ULINT:
		pULint := Value.pValue;
		F_Generic_To_LREAL := TO_LREAL(pULint^);
		
   __SYSTEM.TYPE_CLASS.TYPE_REAL:
		pReal := Value.pValue;
		F_Generic_To_LREAL := TO_LREAL(pReal^);
		
    __SYSTEM.TYPE_CLASS.TYPE_LREAL:
		pLReal := Value.pValue;
		F_Generic_To_LREAL := TO_LREAL(pLReal^);
		
    __SYSTEM.TYPE_CLASS.TYPE_STRING:
		pString := Value.pValue;
		F_Generic_To_LREAL := TO_LREAL(pString^);
		
   __SYSTEM.TYPE_CLASS.TYPE_WSTRING:
		pWString := Value.pValue;
		F_Generic_To_LREAL := TO_LREAL(pWString^);
		
    __SYSTEM.TYPE_CLASS.TYPE_TIME:
		pTime := Value.pValue;
		F_Generic_To_LREAL := TO_LREAL(pTime^);
		
    __SYSTEM.TYPE_CLASS.TYPE_DATE:
		pDate := Value.pValue;
		F_Generic_To_LREAL := TO_LREAL(pDate^);
		
    __SYSTEM.TYPE_CLASS.TYPE_DATEANDTIME:
		pDate_And_Time := Value.pValue;
		F_Generic_To_LREAL := TO_LREAL(pDate_And_Time^);
		
    __SYSTEM.TYPE_CLASS.TYPE_TIMEOFDAY:
		pTime_Of_Day := Value.pValue;
		F_Generic_To_LREAL := TO_LREAL(pTime_Of_Day^);
	
	__SYSTEM.TYPE_CLASS.TYPE_POINTER:
		F_Generic_To_LREAL := TO_LREAL(Value.pValue);
		
	__SYSTEM.TYPE_CLASS.TYPE_LTIME:
		pLTime := Value.pValue;
		F_Generic_To_LREAL := TO_LREAL(pLTime^);
ELSE
	Error := GVL_Errors.ERR_TYPE_MISMATCH;
	RETURN;
	END_CASE

bSuccess := TRUE;

END_FUNCTION

// POUs/Functions/F_Is_Time_Generic
// Checks if a generic is time.
FUNCTION F_Is_Time_Generic : BOOL
VAR_INPUT
	Value : T_Generic;
END_VAR
VAR
END_VAR

CASE Value.TypeClass OF
	__SYSTEM.TYPE_CLASS.TYPE_TIME,
	__SYSTEM.TYPE_CLASS.TYPE_LTIME,
	__SYSTEM.TYPE_CLASS.TYPE_TIMEOFDAY:
		F_Is_Time_Generic := TRUE;
END_CASE

END_FUNCTION

// POUs/Functions/F_Generic_To_LTIME
FUNCTION F_Generic_To_LTIME : LTIME
VAR_INPUT
	 Value : T_Generic;
END_VAR
VAR_OUTPUT
	bSuccess : BOOL;
	Error : T_Error := GVL_Errors.ERR_NO_ERROR;
END_VAR
VAR	
	pBool			: POINTER TO BOOL;
    pByte			: POINTER TO BYTE;
    pWord			: POINTER TO WORD;
    pDWord			: POINTER TO DWORD;
    pLWord			: POINTER TO LWORD;
    pSint			: POINTER TO SINT;
    pInt			: POINTER TO INT;
    pDint			: POINTER TO DINT;
    pLint			: POINTER TO LINT;
    pUSint			: POINTER TO USINT;
    pUInt			: POINTER TO UINT;
    pUDint			: POINTER TO UDINT;
    pULint			: POINTER TO ULINT;
    pReal			: POINTER TO REAL;
    pLReal			: POINTER TO LREAL;
    pString			: POINTER TO STRING(255);
    pWString		: POINTER TO WSTRING;
    pTime			: POINTER TO TIME;
    pDate			: POINTER TO DATE;
    pDate_And_Time	: POINTER TO DATE_AND_TIME;
    pTime_Of_Day	: POINTER TO TIME_OF_DAY;
    pPointer		: PVOID;
	pLTime 			: POINTER TO LTIME;
END_VAR

IF Value.pValue = 0 THEN 
	Error := GVL_Errors.ERR_INVALID_REFERENCE;
	RETURN;
	END_IF;

CASE Value.TypeClass OF 
	__SYSTEM.TYPE_CLASS.TYPE_BOOL:
		pBool := Value.pValue;
		F_Generic_To_LTIME := TO_LTIME(pBool^);
		
    __SYSTEM.TYPE_CLASS.TYPE_BYTE:
		pByte := Value.pValue;
		F_Generic_To_LTIME := TO_LTIME(pByte^);
		
    __SYSTEM.TYPE_CLASS.TYPE_WORD:
		pWord := Value.pValue;
		F_Generic_To_LTIME := TO_LTIME(pWord^);
		
    __SYSTEM.TYPE_CLASS.TYPE_DWORD:
		pDWord := Value.pValue;
		F_Generic_To_LTIME := TO_LTIME(pDWord^);
		
    __SYSTEM.TYPE_CLASS.TYPE_LWORD:
		pLWord := Value.pValue;
		F_Generic_To_LTIME := TO_LTIME(pLWord^);
		
    __SYSTEM.TYPE_CLASS.TYPE_SINT:
		pSint := Value.pValue;
		F_Generic_To_LTIME := TO_LTIME(pSint^);
		
    __SYSTEM.TYPE_CLASS.TYPE_INT:
		pInt := Value.pValue;
		F_Generic_To_LTIME := TO_LTIME(pInt^);
		
    __SYSTEM.TYPE_CLASS.TYPE_DINT:
		pDint := Value.pValue;
		F_Generic_To_LTIME := TO_LTIME(pDint^);
		
    __SYSTEM.TYPE_CLASS.TYPE_LINT:
		pLint := Value.pValue;
		F_Generic_To_LTIME := TO_LTIME(pLint^);
		
    __SYSTEM.TYPE_CLASS.TYPE_USINT:
		pUSint := Value.pValue;
		F_Generic_To_LTIME := TO_LTIME(pUSint^);
		
    __SYSTEM.TYPE_CLASS.TYPE_UINT:
		pUInt := Value.pValue;
		F_Generic_To_LTIME := TO_LTIME(pUInt^);
		
    __SYSTEM.TYPE_CLASS.TYPE_UDINT:
		pUDint := Value.pValue;
		F_Generic_To_LTIME := TO_LTIME(pUDint^);
		
    __SYSTEM.TYPE_CLASS.TYPE_ULINT:
		pULint := Value.pValue;
		F_Generic_To_LTIME := TO_LTIME(pULint^);
		
   __SYSTEM.TYPE_CLASS.TYPE_REAL:
		pReal := Value.pValue;
		F_Generic_To_LTIME := TO_LTIME(pReal^);
		
    __SYSTEM.TYPE_CLASS.TYPE_LREAL:
		pLReal := Value.pValue;
		F_Generic_To_LTIME := TO_LTIME(pLReal^);
		
    __SYSTEM.TYPE_CLASS.TYPE_STRING:
		pString := Value.pValue;
		F_Generic_To_LTIME := TO_LTIME(pString^);
		
   __SYSTEM.TYPE_CLASS.TYPE_WSTRING:
		pWString := Value.pValue;
		F_Generic_To_LTIME := TO_LTIME(pWString^);
		
    __SYSTEM.TYPE_CLASS.TYPE_TIME:
		pTime := Value.pValue;
		F_Generic_To_LTIME := TO_LTIME(pTime^);
		
    __SYSTEM.TYPE_CLASS.TYPE_DATE:
		pDate := Value.pValue;
		F_Generic_To_LTIME := TO_LTIME(pDate^);
		
    __SYSTEM.TYPE_CLASS.TYPE_DATEANDTIME:
		pDate_And_Time := Value.pValue;
		F_Generic_To_LTIME := TO_LTIME(pDate_And_Time^);
		
    __SYSTEM.TYPE_CLASS.TYPE_TIMEOFDAY:
		pTime_Of_Day := Value.pValue;
		F_Generic_To_LTIME := TO_LTIME(TO_TIME(pTime_Of_Day^));
	
	__SYSTEM.TYPE_CLASS.TYPE_POINTER:
		F_Generic_To_LTIME := TO_LTIME(Value.pValue);
		
	__SYSTEM.TYPE_CLASS.TYPE_LTIME:
		pLTime := Value.pValue;
		F_Generic_To_LTIME := TO_LTIME(pLTime^);
ELSE
	Error := GVL_Errors.ERR_TYPE_MISMATCH;
	RETURN;
	END_CASE

bSuccess := TRUE;

END_FUNCTION

// POUs/Functions/F_Is_Date_Generic
// Checks if a generic is a date.
FUNCTION F_Is_Date_Generic : BOOL
VAR_INPUT
	Value : T_Generic;
END_VAR
VAR
END_VAR

CASE Value.TypeClass OF
	__SYSTEM.TYPE_CLASS.TYPE_DATE,
	__SYSTEM.TYPE_CLASS.TYPE_DATEANDTIME:
		F_Is_Date_Generic := TRUE;
END_CASE

END_FUNCTION

// POUs/Functions/F_Generic_To_DT
FUNCTION F_Generic_To_DT : DT
VAR_INPUT
	 Value : T_Generic;
END_VAR
VAR_OUTPUT
	bSuccess : BOOL;
	Error : T_Error := GVL_Errors.ERR_NO_ERROR;
END_VAR
VAR	
	pBool			: POINTER TO BOOL;
    pByte			: POINTER TO BYTE;
    pWord			: POINTER TO WORD;
    pDWord			: POINTER TO DWORD;
    pLWord			: POINTER TO LWORD;
    pSint			: POINTER TO SINT;
    pInt			: POINTER TO INT;
    pDint			: POINTER TO DINT;
    pLint			: POINTER TO LINT;
    pUSint			: POINTER TO USINT;
    pUInt			: POINTER TO UINT;
    pUDint			: POINTER TO UDINT;
    pULint			: POINTER TO ULINT;
    pReal			: POINTER TO REAL;
    pLReal			: POINTER TO LREAL;
    pString			: POINTER TO STRING(255);
    pWString		: POINTER TO WSTRING;
    pTime			: POINTER TO TIME;
    pDate			: POINTER TO DATE;
    pDate_And_Time	: POINTER TO DATE_AND_TIME;
    pTime_Of_Day	: POINTER TO TIME_OF_DAY;
    pPointer		: PVOID;
	pLTime 			: POINTER TO LTIME;
END_VAR

IF Value.pValue = 0 THEN
	Error := GVL_Errors.ERR_INVALID_REFERENCE;
	RETURN;
	END_IF;

CASE Value.TypeClass OF 
	__SYSTEM.TYPE_CLASS.TYPE_BOOL:
		pBool := Value.pValue;
		F_Generic_To_DT := TO_DT(pBool^);
		
    __SYSTEM.TYPE_CLASS.TYPE_BYTE:
		pByte := Value.pValue;
		F_Generic_To_DT := TO_DT(pByte^);
		
    __SYSTEM.TYPE_CLASS.TYPE_WORD:
		pWord := Value.pValue;
		F_Generic_To_DT := TO_DT(pWord^);
		
    __SYSTEM.TYPE_CLASS.TYPE_DWORD:
		pDWord := Value.pValue;
		F_Generic_To_DT := TO_DT(pDWord^);
		
    __SYSTEM.TYPE_CLASS.TYPE_LWORD:
		pLWord := Value.pValue;
		F_Generic_To_DT := TO_DT(pLWord^);
		
    __SYSTEM.TYPE_CLASS.TYPE_SINT:
		pSint := Value.pValue;
		F_Generic_To_DT := TO_DT(pSint^);
		
    __SYSTEM.TYPE_CLASS.TYPE_INT:
		pInt := Value.pValue;
		F_Generic_To_DT := TO_DT(pInt^);
		
    __SYSTEM.TYPE_CLASS.TYPE_DINT:
		pDint := Value.pValue;
		F_Generic_To_DT := TO_DT(pDint^);
		
    __SYSTEM.TYPE_CLASS.TYPE_LINT:
		pLint := Value.pValue;
		F_Generic_To_DT := TO_DT(pLint^);
		
    __SYSTEM.TYPE_CLASS.TYPE_USINT:
		pUSint := Value.pValue;
		F_Generic_To_DT := TO_DT(pUSint^);
		
    __SYSTEM.TYPE_CLASS.TYPE_UINT:
		pUInt := Value.pValue;
		F_Generic_To_DT := TO_DT(pUInt^);
		
    __SYSTEM.TYPE_CLASS.TYPE_UDINT:
		pUDint := Value.pValue;
		F_Generic_To_DT := TO_DT(pUDint^);
		
    __SYSTEM.TYPE_CLASS.TYPE_ULINT:
		pULint := Value.pValue;
		F_Generic_To_DT := TO_DT(pULint^);
		
   __SYSTEM.TYPE_CLASS.TYPE_REAL:
		pReal := Value.pValue;
		F_Generic_To_DT := TO_DT(pReal^);
		
    __SYSTEM.TYPE_CLASS.TYPE_LREAL:
		pLReal := Value.pValue;
		F_Generic_To_DT := TO_DT(pLReal^);
		
    __SYSTEM.TYPE_CLASS.TYPE_STRING:
		pString := Value.pValue;
		F_Generic_To_DT := TO_DT(pString^);
		
   __SYSTEM.TYPE_CLASS.TYPE_WSTRING:
		pWString := Value.pValue;
		F_Generic_To_DT := TO_DT(pWString^);
		
    __SYSTEM.TYPE_CLASS.TYPE_TIME:
		pTime := Value.pValue;
		F_Generic_To_DT := TO_DT(pTime^);
		
    __SYSTEM.TYPE_CLASS.TYPE_DATE:
		pDate := Value.pValue;
		F_Generic_To_DT := TO_DT(pDate^);
		
    __SYSTEM.TYPE_CLASS.TYPE_DATEANDTIME:
		pDate_And_Time := Value.pValue;
		F_Generic_To_DT := TO_DT(pDate_And_Time^);
		
    __SYSTEM.TYPE_CLASS.TYPE_TIMEOFDAY:
		pTime_Of_Day := Value.pValue;
		F_Generic_To_DT := TO_DT(pTime_Of_Day^);
	
	__SYSTEM.TYPE_CLASS.TYPE_POINTER:
		F_Generic_To_DT := TO_DT(Value.pValue);
		
	__SYSTEM.TYPE_CLASS.TYPE_LTIME:
		pLTime := Value.pValue;
		F_Generic_To_DT := TO_DT(pLTime^);
ELSE
	Error := GVL_Errors.ERR_TYPE_MISMATCH;
	RETURN;
	END_CASE

bSuccess := TRUE;

END_FUNCTION

// POUs/Functions/F_Clone_Generic
// Clones a generic.
// NOTE: memory is allocated in the heap for the clone and is set to pValue. Dont forget to delete it when done. 
FUNCTION F_Clone_Generic : T_Generic
VAR_INPUT
	Source : T_Generic;
END_VAR
VAR_OUTPUT
	bSuccess : BOOL;
	Error : T_Error := GVL_Errors.ERR_NO_ERROR;
END_VAR

F_Clone_Generic.diSize := Source.diSize;
F_Clone_Generic.TypeClass := Source.TypeClass;

IF Source.pValue = 0 OR_ELSE Source.diSize = 0 THEN bSuccess := TRUE; RETURN; END_IF

F_Clone_Generic.pValue := __NEW(BYTE, TO_UDINT(Source.diSize));

IF F_Clone_Generic.pValue = 0 THEN
	Error := GVL_Errors.ERR_MALLOC_FAILED;
	RETURN;
	END_IF

CASE Source.TypeClass OF
	T_Type.TYPE_STRING:
		Tc2_Utilities.STRNCPY(F_Clone_Generic.pValue, Source.pValue, TO_UDINT(Source.diSize));
	T_Type.TYPE_WSTRING:
		Tc2_Utilities.WSTRNCPY(F_Clone_Generic.pValue, Source.pValue, TO_UDINT(Source.diSize));
ELSE
	Tc2_System.MEMCPY(F_Clone_Generic.pValue, Source.pValue, TO_UDINT(Source.diSize));
	END_CASE
	
bSuccess := TRUE;

END_FUNCTION

// POUs/Function Blocks/Collections/FB_Array_List
// A dynamic array that can grow and shrink as needed..
{attribute 'enable_dynamic_creation'}
{attribute 'no_assign'}
{attribute 'no_explicit_call' := 'direct call for this function block is not allowed'}
FUNCTION_BLOCK FB_Array_List EXTENDS FB_Collection IMPLEMENTS I_Array_List, I_Iterable//, I_Enumerable, I_Copyable
VAR
	pBuffer : POINTER TO T_Generic;
	Capacity : T_Capacity;
END_VAR

// Index of the first element.
PROPERTY _Begin : T_Position
GET
_Begin := 0;
END_GET
END_PROPERTY

// Size of the storage space currently allocated for the array list.
PROPERTY FINAL _Capacity : T_Capacity
GET
_Capacity := THIS^.Capacity;
END_GET
SET
PROTECTED 
VAR
END_VAR
THIS^.Capacity := _Capacity;
END_SET
END_PROPERTY

// Index of the last element.
PROPERTY _End : T_Position
GET
_End := TO_DINT(THIS^._Count) - 1;
END_GET
END_PROPERTY

// Adds an item to the end of the list.
METHOD Append : I_List
VAR_INPUT
	Item : ANY; // Value to store in list
END_VAR
VAR_OUTPUT
	bSuccess : BOOL;
END_VAR
Append := THIS^;

THIS^.Insert_Generic(THIS^._Count, Item, bSuccess => bSuccess);
END_METHOD

// Empties/Clears/Deletes every item in the list.
METHOD Clear : I_List
VAR
	i : T_Capacity;
END_VAR
Clear := THIS^;

THIS^.Clear_Error();

IF THIS^.pBuffer = 0 OR_ELSE THIS^._Empty THEN RETURN; END_IF

FOR i := 0 TO THIS^._Count - 1 DO
	F_Delete_Generic(THIS^.pBuffer[i]);
	END_FOR
	
THIS^._Count := 0;
END_METHOD

// Checks if item is contained in list.
METHOD Contains : BOOL
VAR_INPUT
	Item : ANY; // Item to find in list
END_VAR
THIS^.Search(Item, bSuccess => Contains);
END_METHOD

{attribute 'hide'}
METHOD FB_exit : BOOL
VAR_INPUT
	bInCopyCode : BOOL; // if TRUE, the exit method is called for exiting an instance that is copied afterwards (online change).
END_VAR
// Return if it's an online change.
IF bInCopyCode OR_ELSE THIS^.pBuffer = 0 THEN RETURN; END_IF

THIS^.Clear();
__DELETE(THIS^.pBuffer);
THIS^._Capacity := 0;
END_METHOD

{attribute 'hide'}
METHOD FB_init : BOOL
VAR_INPUT
	bInitRetains 		: BOOL; // if TRUE, the retain variables are initialized (warm start / cold start)
	bInCopyCode 		: BOOL; // if TRUE, the instance afterwards gets moved into the copy code (online change)
	Initial_Capacity 	: T_Capacity; // The capacity and count to initialise the array list with.
END_VAR
VAR 
	i : T_Capacity;
END_VAR
// Return if it's an online change.
IF bInCopyCode THEN RETURN; END_IF

THIS^.Resize(Initial_Capacity);
THIS^._Count := THIS^._Capacity;
END_METHOD

// Gets item from list at specified location without removing it
METHOD Get : I_List
VAR_INPUT
	Index : T_Position; // Location of item
	Item : ANY;  // Variable to store returned item
END_VAR
VAR_OUTPUT
	bSuccess : BOOL;
END_VAR
Get := THIS^;

IF Index < 0 OR_ELSE Index >= THIS^._Count THEN
	THIS^._Error_Status := GVL_Errors.ERR_INDEX_OUT_OF_BOUNDS;
	RETURN;
	END_IF

IF NOT F_Matching_Generics(Item, THIS^.pBuffer[Index]) THEN
	THIS^._Error_Status := GVL_Errors.ERR_TYPE_MISMATCH;
	RETURN;
	END_IF
	
F_Copy_Generic_Value(THIS^.pBuffer[Index], Item, bSuccess => bSuccess, Error => THIS^.Error);
END_METHOD

// Returns item as a string, if type to string conversion is supported
METHOD Get_As_String : I_List
VAR_INPUT
	Index : T_Position; // Location of item
	sItem : REFERENCE TO STRING; // Variable to store returned item.
END_VAR
VAR_OUTPUT
	bSuccess : BOOL;
END_VAR
Get_As_String := THIS^;

IF NOT __ISVALIDREF(sItem) THEN 
	THIS^._Error_Status := GVL_Errors.ERR_INVALID_REFERENCE;
	RETURN;
	END_IF

IF Index < 0 OR_ELSE Index >= THIS^._Count THEN
	THIS^._Error_Status := GVL_Errors.ERR_INDEX_OUT_OF_BOUNDS;
	RETURN;
	END_IF
	
CASE THIS^.pBuffer[Index].TypeClass OF
	T_Type.TYPE_STRING:
		Tc2_Utilities.STRNCPY(ADR(sItem), THIS^.pBuffer[Index].pValue, MIN(Tc2_Utilities.LEN2(ADR(sItem))+1, TO_UDINT(THIS^.pBuffer[Index].diSize)));
		THIS^.Clear_Error();

	T_Type.TYPE_WSTRING:
		Tc2_Utilities.WSTRING_TO_STRING2(ADR(sItem), THIS^.pBuffer[Index].pValue, MIN(Tc2_Utilities.LEN2(ADR(sItem))+1, TO_UDINT(THIS^.pBuffer[Index].diSize)));
		THIS^.Clear_Error();
ELSE
	sItem := F_Generic_To_String(THIS^.pBuffer[Index], bSuccess => bSuccess, Error => THIS^.Error);
	END_CASE
END_METHOD

// Gets a value from a list in it's generic form.
// (** Use carefully as this contains the pointer of the actual value in the collection. **)
// If you wish to use this it is recommeded you create a copy of the returned value using MEMMOVE or MEMCPY
METHOD Get_Generic : I_List
VAR_INPUT
	Index : T_Position; // Location of item
END_VAR
VAR_OUTPUT
	Item : T_Generic := (TypeClass := T_Type.TYPE_NONE);
	bSuccess : BOOL;
END_VAR
Get_Generic := THIS^;

IF Index < 0 OR_ELSE Index >= THIS^._Count THEN
	THIS^._Error_Status := GVL_Errors.ERR_INDEX_OUT_OF_BOUNDS;
	RETURN;
	END_IF

Item := THIS^.pBuffer[Index];
bSuccess := TRUE;
THIS^.Clear_Error();
END_METHOD

// Gets the type of the item at specified location.
METHOD Get_Type_At : I_List
VAR_INPUT
	Index : T_Position;
END_VAR
VAR_OUTPUT
	Item_Type : T_Type := T_Type.TYPE_NONE;
	bSuccess : BOOL;
END_VAR
VAR
	Tmp : T_Generic;
END_VAR
Get_Type_At := THIS^;

THIS^.Get_Generic(Index, Item => Tmp, bSuccess => bSuccess);

IF bSuccess THEN Item_Type := Tmp.TypeClass; END_IF
END_METHOD

// Adds new item to list at specified location, if index = 0, item will be added at the front, if index = count, item will be added at the back
METHOD Insert : I_List
VAR_INPUT
	Index : T_Position; // Location of item
	Item : ANY; // Item to store in list
END_VAR
VAR_OUTPUT
	bSuccess : BOOL;
END_VAR
Insert := THIS^;
THIS^.Insert_Generic(Index, Item, bSuccess => bSuccess);
END_METHOD

// Adds new item to list at specified location using the generic form. 
// If index = 0, item will be added at the front, if index = count, item will be added at the back
METHOD Insert_Generic : I_List
VAR_INPUT
	Index 	 : T_Position; 	// Location of item
	Item 	 : T_Generic;  	// Item to store in list
END_VAR
VAR_OUTPUT
	bSuccess : BOOL;
END_VAR
VAR 
	Tmp : T_Generic;
END_VAR
Insert_Generic := THIS^;

IF THIS^._Count >= THIS^._Capacity THEN 
	// Increase capacity by 50% if it's greater than 1 else change to 16.
	THIS^.Resize(SEL(THIS^._Count > 1, 16, THIS^._Count + SHR(THIS^._Count, 1)), bSuccess => bSuccess);
	IF NOT bSuccess THEN RETURN; END_IF
	END_IF

IF Index = THIS^._Count THEN 
	// Add to back.
	Tmp := F_Clone_Generic(Item, bSuccess => bSuccess, Error => THIS^.Error);
	IF NOT bSuccess THEN RETURN; END_IF
	THIS^.pBuffer[THIS^._Count] := Tmp;
	THIS^.Increment_Count();
	RETURN;
	END_IF

IF Index < 0 OR_ELSE Index > THIS^._Count THEN
	// Throw out of bounds error.
	THIS^._Error_Status := GVL_Errors.ERR_INDEX_OUT_OF_BOUNDS;
	bSuccess := FALSE;
	RETURN;
	END_IF

Tmp := F_Clone_Generic(Item, bSuccess => bSuccess, Error => Error);
IF NOT bSuccess THEN RETURN; END_IF

Tc2_System.MEMMOVE(ADR(THIS^.pBuffer[Index + 1]), ADR(THIS^.pBuffer[Index]), TO_UDINT((THIS^._Count - Index) * SIZEOF(T_Generic)));
THIS^.pBuffer[Index] := Tmp;
THIS^.Increment_Count();
END_METHOD

// Adds an item at the front of the list.
METHOD Prepend : I_List
VAR_INPUT
	Item : ANY; // Value to store in list
END_VAR
VAR_OUTPUT
	bSuccess : BOOL;
END_VAR
Prepend := THIS^;

THIS^.Insert_Generic(0, Item, bSuccess => bSuccess);
END_METHOD

// Removes item from the list.
METHOD Remove : I_List
VAR_INPUT
	Item : ANY; // Item to remove from in list
END_VAR
VAR_OUTPUT
	bSuccess : BOOL;
END_VAR
VAR
	Tmp : T_Position := -1;
END_VAR
Remove := THIS^;

THIS^.Search(Item, Index => Tmp, bSuccess => bSuccess);
IF NOT bSuccess THEN RETURN; END_IF 
THIS^.Remove_At(Tmp, bSuccess => bSuccess);
END_METHOD

// Remove item at specified location 
METHOD Remove_At : I_List
VAR_INPUT
	Index : T_Position; // Location of item
END_VAR
VAR_OUTPUT
	bSuccess : BOOL;
END_VAR
Remove_At := THIS^;

IF Index < 0 OR_ELSE Index >= THIS^._Count THEN
	THIS^._Error_Status := GVL_Errors.ERR_INDEX_OUT_OF_BOUNDS;
	RETURN;
	END_IF

F_Delete_Generic(THIS^.pBuffer[Index]);	
Tc2_System.MEMMOVE(ADR(THIS^.pBuffer[Index]), ADR(THIS^.pBuffer[Index+1]), TO_UDINT(SIZEOF(T_Generic)*(THIS^._Count - Index - 1)));
THIS^.Decrement_Count();

IF THIS^._Count <= (THIS^._Capacity/4) THEN THIS^.Resize(THIS^._Capacity/2); END_IF

bSuccess := TRUE;
THIS^.Clear_Error();
END_METHOD

// Removes item at the back of the list.
METHOD Remove_Last : I_List
VAR_OUTPUT
	bSuccess : BOOL;
END_VAR
Remove_Last := THIS^.Remove_At(THIS^._Count - 1, bSuccess => bSuccess);
END_METHOD

// Manually resize list. If list becomes smaller, item on higher locations will be deleted.
METHOD Resize : I_List
VAR_INPUT
	Size : T_Capacity; // New size of list.
END_VAR
VAR_OUTPUT
	bSuccess : BOOL;
END_VAR
VAR
	pNew_Buffer : POINTER TO T_Generic;
	i, Number_Of_Elements_To_Copy : T_Capacity;
END_VAR
Resize := THIS^;

IF Size = 0 THEN THIS^.FB_exit(FALSE); bSuccess := TRUE; RETURN; END_IF
IF THIS^.pBuffer = 0 THEN 
	THIS^.pBuffer := F_Malloc_Generic(1, bSuccess => bSuccess, Error => THIS^.Error);
	IF NOT bSuccess THEN RETURN; END_IF
	THIS^._Capacity := 1;
	END_IF

pNew_Buffer := F_Malloc_Generic(Size, bSuccess => bSuccess, Error => THIS^.Error);
IF NOT bSuccess THEN RETURN; END_IF

Tc2_System.MEMCPY(pNew_Buffer, THIS^.pBuffer, TO_UDINT(SIZEOF(T_Generic)*THIS^._Count));

IF Size < THIS^._Count THEN
	FOR i := Size TO THIS^._Count - 1 DO F_Delete_Generic(THIS^.pBuffer[i]); END_FOR
	THIS^._Count := Size;
	END_IF

THIS^._Capacity := Size;

__DELETE(THIS^.pBuffer);
THIS^.pBuffer := pNew_Buffer;
END_METHOD

// Reverses the order of items in the list
METHOD Reverse : I_List
VAR_OUTPUT
	bSuccess : BOOL;
END_VAR
VAR
	i : T_Capacity;
END_VAR
Reverse := THIS^;

IF NOT THIS^._Empty THEN
	FOR i := 0 TO (THIS^._Count/2) - 1 DO
		F_Swap_Generics(THIS^.pBuffer[i], THIS^.pBuffer[THIS^._Count - i - 1]);
		END_FOR
	END_IF

bSuccess := TRUE;
THIS^.Clear_Error();
END_METHOD

// Find the location of an item in list.
METHOD Search : I_List
VAR_INPUT
	Item : ANY; // Item to find in list
END_VAR
VAR_OUTPUT
	Index : T_Position := -1; //Location of item in list 
	bSuccess : BOOL;
END_VAR
VAR
	i : T_Position;
END_VAR
Search := THIS^;

IF THIS^._Empty THEN RETURN; END_IF
FOR i := 0 TO THIS^._Count - 1 DO
	CASE F_Compare_Generics(Item, THIS^.pBuffer[i]) OF
		T_Comparison.Equal:
			bSuccess := TRUE;
			THIS^.Clear_Error();
			Index := i;
			RETURN;
		END_CASE
	END_FOR
	
THIS^._Error_Status := GVL_Errors.ERR_NO_ITEM;
END_METHOD

// Changes the item at the specified location in the list.
METHOD Set : I_List
VAR_INPUT
	Index 	: T_Position; // Location of item
	Item 	: ANY; 	// Item to store in list
END_VAR
VAR_OUTPUT
	bSuccess : BOOL;
END_VAR
Set := THIS^;

THIS^.Set_Generic(Index, Item, bSuccess => bSuccess);
END_METHOD

// Changes the item at the specified location in the list in it's generic form.
METHOD Set_Generic : I_List
VAR_INPUT
	Index : T_Position; // Location of item
	Item : T_Generic;
END_VAR
VAR_OUTPUT
	bSuccess : BOOL;
END_VAR
VAR
	Tmp : T_Generic;
END_VAR
Set_Generic := THIS^;

IF Index < 0 OR_ELSE Index >= THIS^._Count THEN
	THIS^._Error_Status := GVL_Errors.ERR_INDEX_OUT_OF_BOUNDS;
	RETURN;
	END_IF
	
Tmp := F_Clone_Generic(Item, bSuccess => bSuccess, Error => THIS^.Error);

IF NOT bSuccess THEN RETURN; END_IF

F_Delete_Generic(THIS^.pBuffer[Index]);

THIS^.pBuffer[Index] := Tmp;
END_METHOD

// Swaps item at index A with item at index B.
METHOD Swap : I_List
VAR_INPUT
	Index_A, Index_B : T_Position;
END_VAR
VAR_OUTPUT
	bSuccess : BOOL;
END_VAR
Swap := THIS^;

IF Index_A < 0 OR_ELSE Index_A >= THIS^._Count OR_ELSE Index_B < 0 OR_ELSE Index_B >= THIS^._Count THEN
	THIS^._Error_Status := GVL_Errors.ERR_INDEX_OUT_OF_BOUNDS;
	RETURN;
	END_IF
	
bSuccess := F_Swap_Generics(THIS^.pBuffer[Index_A], THIS^.pBuffer[Index_B], bSuccess => bSuccess, Error => THIS^.Error);
END_METHOD

END_FUNCTION_BLOCK

// POUs/Function Blocks/Collections/FB_Deque
// (Pronounced Deck) Double ended queue. A collection that supports the insertion and removal of items at the front and back.
{attribute 'enable_dynamic_creation'}
{attribute 'no_assign'}
{attribute 'no_explicit_call' := 'direct call for this function block is not allowed'}
FUNCTION_BLOCK FB_Deque IMPLEMENTS I_Deque//, I_Enumerable, I_Copyable
VAR
	fbList : FB_List := ();
END_VAR

// Number of items in the collection.
PROPERTY _Count : T_Capacity
GET
_Count := THIS^.fbList._Count;
END_GET
END_PROPERTY

// Checks if collection is empty.
PROPERTY _Empty : BOOL
GET
_Empty := THIS^.fbList._Empty;
END_GET
END_PROPERTY

// Error status of the collection.
PROPERTY _Error_Status : T_Error
GET
_Error_Status := THIS^.fbList._Error_Status;
END_GET
END_PROPERTY

// Gets an immutable list of the items in Deque.
PROPERTY _Values : I_Immutable_List
GET
VAR_INST
	fbImmutable_List : FB_Immutable_List := (ipList := THIS^.fbList);
END_VAR
_Values := fbImmutable_List;
END_GET
END_PROPERTY

// Get item at the back of the deque without removing it.
METHOD Back : I_Deque
VAR_INPUT
	Item : ANY; // Variable to store returned item value
END_VAR
VAR_OUTPUT
	bSuccess : BOOL;
END_VAR
Back := THIS^;

THIS^.fbList.Get(THIS^.fbList._Count - 1, Item, bSuccess => bSuccess);
END_METHOD

// Empties/Clears/Deletes every item in the deque.
METHOD Clear : I_Deque
Clear := THIS^;

THIS^.fbList.Clear();
END_METHOD

// Removes item at the front of the deque.
METHOD Dequeue_At_Back : I_Deque
VAR_OUTPUT
	bSuccess : BOOL;
END_VAR
Dequeue_At_Back := THIS^;

THIS^.fbList.Remove_Last(bSuccess => bSuccess);
END_METHOD

// Removes item at the front of the deque.
METHOD Dequeue_At_Front : I_Deque
VAR_OUTPUT
	bSuccess : BOOL;
END_VAR
Dequeue_At_Front := THIS^;

THIS^.fbList.Remove_At(0, bSuccess => bSuccess);
END_METHOD

// Adds item at the back of the deque.
METHOD Enqueue_At_Back : I_Deque
VAR_INPUT
	Item : ANY; // Item to store.
END_VAR
VAR_OUTPUT
	bSuccess : BOOL;
END_VAR
Enqueue_At_Back := THIS^.Enqueue_Generic(Item, FALSE,bSuccess => bSuccess);
END_METHOD

// Add item to the front of the deque.
METHOD Enqueue_At_Front : I_Deque
VAR_INPUT
	Item : ANY; // Item to store.
END_VAR
VAR_OUTPUT
	bSuccess : BOOL;
END_VAR
Enqueue_At_Front := THIS^.Enqueue_Generic(Item, TRUE,bSuccess => bSuccess);
END_METHOD

